// ---- POUs/Logic/Sequencing/Permissives/FB_Permissives.TcPOU
(*
PERMISSIVE - Operational Enabling Function Block
================================================
Philosophy: Allows a change in state only when all conditions are met.
Behavior:   Follows real-time conditions, no latching, can be bypassed for
            maintenance.
Logic:      Mapped bits 1 = good, 0 = bad. Unmapped bits default good (1).
            sts.bOK = TRUE when every active permissive bit is good (or
            bypassed). Non-latching: status tracks real-time inputs.
Mapping:    Call MapInput(bitIndex, value) every cycle for each active
            permissive. Unmapped bits automatically reset to good after
            FB_BitMatrix64's MAPPING_TIMEOUT cycles.

The 64-bit condition-matrix machinery is shared with FB_Interlock via
FB_BitMatrix64 — the difference between the two FBs is latching semantics,
which lives here (or in FB_Interlock) on top of the shared core.
*)
{attribute 'OPC.UA.DA' := '1'}
FUNCTION_BLOCK PUBLIC FB_Permissives
VAR_INPUT
    {attribute 'OPC.UA.DA' := '1'}
    {attribute 'OPC.UA.DA.Access' := '1'}
    cfg : ST_Permissive_Config;
END_VAR
VAR_OUTPUT
    {attribute 'OPC.UA.DA' := '1'}
    {attribute 'OPC.UA.DA.Access' := '1'}
    sts : ST_Permissive_Status;
END_VAR
VAR
    {attribute 'OPC.UA.DA' := '0'}
    _core : FB_BitMatrix64;
END_VAR

// Drive the shared bit-matrix machinery (cycle counter, cleanup, transitions).
_core.ConstrainBypass(allowedMask := cfg.nBypassable);
_core();

// Non-latching rollup: unmapped bits default good, bypassed bits forced good.
sts.nPermissives          := (_core.nLiveBits OR NOT _core.nActiveMask) OR _core.nBypassMask;
sts.nBypassMask           := _core.nBypassMask;
sts.nFirstFailureBitIndex := _core.nFirstFailureBitIndex;
sts.bOK                   := sts.nPermissives = 16#FFFFFFFFFFFFFFFF;

sts.nMissing := cfg.nRequired AND NOT _core.nActiveMask;
sts.nPermissives := sts.nPermissives AND NOT sts.nMissing;
sts.bOK := sts.bOK AND (sts.nMissing = 0);
UpdateFaceplates();

(*
Map a boolean signal to one permissive bit (0..63). TRUE = good, FALSE = bad.
Call every cycle for each active permissive condition.
*)
METHOD PUBLIC MapInput
VAR_INPUT
    bitIndex   : UDINT;
    inputValue : BOOL;
END_VAR
_core.MapInput(bitIndex := bitIndex, inputValue := inputValue);
END_METHOD

(*
Reset - Clear all bypass states. Permissives follow real-time conditions
(non-latching) so there is nothing else to clear.
*)
METHOD Reset
_core.ClearBypass();
END_METHOD

(*
Set or clear bypass for a specific permissive bit. Only bits configured
as bypassable in cfg.nBypassable can be enabled; clearing is always allowed.
*)
METHOD PUBLIC SetBypass : E_RpcMethodResponse
VAR_INPUT
    bitIndex : UDINT;
    bEnable  : BOOL;
END_VAR
SetBypass := _core.SetBypass(
    bitIndex        := bitIndex,
    bEnable         := bEnable,
    nBypassableMask := cfg.nBypassable);
END_METHOD

METHOD PRIVATE UpdateFaceplates
VAR
    i       : UDINT;
    bitMask : ULINT;
END_VAR
FOR i := 0 TO 63 DO
    bitMask := SHL(ULINT#1, i);
    sts.aFaceplates[i].name          := cfg.aNames[i];
    sts.aFaceplates[i].ok         := (sts.nPermissives AND bitMask) <> 0;
    sts.aFaceplates[i].mapped     := (_core.nActiveMask AND bitMask) <> 0;
    sts.aFaceplates[i].bypassed   := (_core.nBypassMask AND bitMask) <> 0;
    sts.aFaceplates[i].bypassable := (cfg.nBypassable  AND bitMask) <> 0;
END_FOR;
END_METHOD

END_FUNCTION_BLOCK

// ---- POUs/Utilities/FB_BitMatrix64.TcPOU
// ============================================================================
// FB_BitMatrix64 — Shared 64-bit condition-matrix core
// ============================================================================
// Internal composition helper used by FB_Permissives (non-latching) and
// FB_Interlock (latching). Encapsulates the mechanics both FBs share:
//
//   - 64 bits of "good (1) / bad (0)" live state fed by MapInput()
//   - an active-mask so unmapped bits default to good and bypass logic is
//     parameterised on the caller's cfg.nBypassable (no cfg coupling here)
//   - cycle-based cleanup that unmaps a bit if it hasn't been re-fed within
//     MAPPING_TIMEOUT scans
//   - first-failure tracking (sequence counter + first-failure bit index)
//   - "just unmapped while bad" events so the caller can latch that memory
//     if it needs to (FB_Interlock.nUnmappedBadBits)
//
// The caller composes an instance, calls the cyclic body, then computes its
// own effective mask / rollup (interlocks latch; permissives don't). See
// docs/2-Architecture.md for the split between the two surfaces.
// ============================================================================
{attribute 'OPC.UA.DA' := '0'}
FUNCTION_BLOCK FB_BitMatrix64
VAR_OUTPUT
    // Current live bits (1=good, 0=bad). Unmapped bits are held at 1.
    nLiveBits             : ULINT := 16#FFFFFFFFFFFFFFFF;
    // 1 = bit is actively mapped (refreshed within MAPPING_TIMEOUT cycles).
    nActiveMask           : ULINT := 0;
    // Dynamic bypass mask (1=bypassed). See SetBypass / ClearBypass.
    nBypassMask           : ULINT := 0;
    // Bit index (0..63) of the first bit to go bad in the current failure
    // sequence; 999 when no sequence is active.
    nFirstFailureBitIndex : UDINT := 999;
    // Bits that transitioned from active to unmapped *this cycle* while
    // their live value was bad. OR'd each cycle; caller latches if it cares.
    nJustUnmappedBad      : ULINT := 0;
END_VAR
VAR
    _previousBits     : ULINT := 16#FFFFFFFFFFFFFFFF;
    _cycleCounter     : UDINT := 0;
    _lastMappedCycle  : ARRAY[0..63] OF UDINT;
    _sequenceCounter  : UDINT := 0;
    MAPPING_TIMEOUT   : UDINT := 10;
END_VAR

_cycleCounter := _cycleCounter + 1;
IF _cycleCounter = 0 THEN _cycleCounter := 1; END_IF;

nJustUnmappedBad := 0;
_CleanupUnmapped();
_DetectTransitions();

_previousBits := nLiveBits;

// Feed one bit's live value. Call every cycle for every active condition;
// any bit not refreshed within MAPPING_TIMEOUT scans is automatically
// considered unmapped and its live bit snaps back to good.
METHOD PUBLIC MapInput
VAR_INPUT
    bitIndex   : UDINT;
    inputValue : BOOL;
END_VAR
VAR
    bitMask : ULINT;
END_VAR
IF bitIndex > 63 THEN RETURN; END_IF;

bitMask := SHL(ULINT#1, bitIndex);
nActiveMask := nActiveMask OR bitMask;
_lastMappedCycle[bitIndex] := _cycleCounter;

IF inputValue THEN
    nLiveBits := nLiveBits OR bitMask;
ELSE
    nLiveBits := nLiveBits AND NOT bitMask;
END_IF;
END_METHOD

// Enable/disable bypass for a single bit. The caller passes its own
// cfg.nBypassable so this FB stays decoupled from caller-specific cfg DUTs.
// Clearing a bypass is always permitted; enabling requires the bit to be
// marked bypassable.
METHOD PUBLIC SetBypass : E_RpcMethodResponse
VAR_INPUT
    bitIndex         : UDINT;
    bEnable          : BOOL;
    nBypassableMask  : ULINT;
END_VAR
VAR
    bitMask : ULINT;
END_VAR
IF bitIndex > 63 THEN
    SetBypass := E_RpcMethodResponse.REJECTED_INVALID_PARAMETER;
    RETURN;
END_IF;

bitMask := SHL(ULINT#1, bitIndex);

IF bEnable AND (nBypassableMask AND bitMask) = 0 THEN
    SetBypass := E_RpcMethodResponse.REJECTED_BYPASS_NOT_ALLOWED;
    RETURN;
END_IF;

IF bEnable THEN
    nBypassMask := nBypassMask OR bitMask;
ELSE
    nBypassMask := nBypassMask AND NOT bitMask;
END_IF;

SetBypass := E_RpcMethodResponse.ACCEPTED;
END_METHOD

// Clear every bypass bit at once (e.g. on a Reset()).
METHOD PUBLIC ClearBypass
nBypassMask := 0;
END_METHOD

// Drop any first-failure sequence in progress.
METHOD PUBLIC ClearFirstFailure
nFirstFailureBitIndex := 999;
_sequenceCounter      := 0;
END_METHOD

METHOD PRIVATE _CleanupUnmapped
VAR
    i       : UDINT;
    bitMask : ULINT;
END_VAR
FOR i := 0 TO 63 DO
    bitMask := SHL(ULINT#1, i);
    IF (nActiveMask AND bitMask) <> 0 THEN
        IF (_cycleCounter - _lastMappedCycle[i]) > MAPPING_TIMEOUT THEN
            // Expose bad-at-unmap as an event so latching callers (FB_Interlock)
            // can remember it. Non-latching callers simply ignore this output.
            IF (nLiveBits AND bitMask) = 0 THEN
                nJustUnmappedBad := nJustUnmappedBad OR bitMask;
            END_IF;
            nActiveMask := nActiveMask AND NOT bitMask;
            nLiveBits   := nLiveBits   OR bitMask;
        END_IF;
    END_IF;
END_FOR;
END_METHOD

METHOD PRIVATE _DetectTransitions
VAR
    i       : UDINT;
    bitMask : ULINT;
END_VAR
// New failure sequence: all-good last cycle, something bad now.
IF _previousBits = 16#FFFFFFFFFFFFFFFF AND nLiveBits <> 16#FFFFFFFFFFFFFFFF THEN
    _sequenceCounter      := 0;
    nFirstFailureBitIndex := 999;
END_IF;

FOR i := 0 TO 63 DO
    bitMask := SHL(ULINT#1, i);
    IF (nActiveMask AND bitMask) <> 0 THEN
        IF ((_previousBits AND bitMask) <> 0) AND ((nLiveBits AND bitMask) = 0) THEN
            _sequenceCounter := _sequenceCounter + 1;
            IF _sequenceCounter = 1 THEN
                nFirstFailureBitIndex := i;
            END_IF;
        END_IF;
    END_IF;
END_FOR;
END_METHOD

// Revocation is permanent; allowing the bit again requires a fresh SetBypass.
METHOD PUBLIC ConstrainBypass
VAR_INPUT allowedMask : ULINT; END_VAR
nBypassMask := nBypassMask AND allowedMask;
END_METHOD

END_FUNCTION_BLOCK

// ---- POUs/Logic/Interlocks/FB_Interlock.TcPOU
(*
INTERLOCK - Safety Protection Function Block
============================================
Philosophy: Prevents unsafe conditions from continuing. Latches bad
            conditions until a deliberate Reset() call, even if the
            real-world condition has already recovered.
Behavior:   Every mapped bit latches by design. Reset() is required to
            clear latched bits. Bypass is available per bit only if
            cfg.nBypassable marks the bit as bypassable.
Logic:      Mapped bits 1 = good, 0 = bad. Unmapped bits default good.
            A bit that was bad at the time its mapping stopped is
            remembered and keeps sts.bOK FALSE until Reset() is called.
            sts.bOK = TRUE when every active interlock bit is good.
Mapping:    Call MapInput(bitIndex, value) every cycle for each active
            interlock condition. Unmapped bits automatically reset to
            good after FB_BitMatrix64's MAPPING_TIMEOUT cycles.
Clearing:   Call Reset() after the real-world conditions have cleared.

The 64-bit condition-matrix machinery is shared with FB_Permissives via
FB_BitMatrix64; the latching + unmapped-bad memory is the interlock-only
logic that sits on top.

Contrast with FB_Permissives: permissives are non-latching operational
readiness checks; interlocks are latching safety protections.
*)
{attribute 'OPC.UA.DA' := '1'}
FUNCTION_BLOCK PUBLIC FB_Interlock
VAR_INPUT
    {attribute 'OPC.UA.DA' := '1'}
    {attribute 'OPC.UA.DA.Access' := '1'}
    cfg : ST_Interlock_Config;
END_VAR
VAR_OUTPUT
    {attribute 'OPC.UA.DA' := '1'}
    {attribute 'OPC.UA.DA.Access' := '1'}
    sts : ST_Interlock_Status;
END_VAR
VAR
    {attribute 'OPC.UA.DA' := '0'}
    _core            : FB_BitMatrix64;
    {attribute 'OPC.UA.DA' := '0'}
    _latchedBits     : ULINT := 16#FFFFFFFFFFFFFFFF;
    {attribute 'OPC.UA.DA' := '0'}
    _unmappedBadBits : ULINT := 0;
END_VAR

// Drive the shared bit-matrix machinery (cycle counter, cleanup, transitions).
_core.ConstrainBypass(allowedMask := cfg.nBypassable);
_core();

// Carry forward any "bad at unmap" memory — keeps sts.bOK FALSE until Reset().
_unmappedBadBits := _unmappedBadBits OR _core.nJustUnmappedBad OR (cfg.nRequired AND NOT _core.nActiveMask);

// Latch once a mapped bit goes bad; inactive/unmapped bits remain good.
_latchedBits := (_latchedBits AND _core.nLiveBits) OR NOT _core.nActiveMask;

// Effective: latched-or-unmapped, then forced good by any bypass bits.
sts.nInterlocks           := (_latchedBits OR NOT _core.nActiveMask) OR _core.nBypassMask;
sts.nLatched              := _latchedBits;
sts.nBypassMask           := _core.nBypassMask;
sts.nFirstFailureBitIndex := _core.nFirstFailureBitIndex;
sts.bOK                   := (sts.nInterlocks = 16#FFFFFFFFFFFFFFFF) AND (_unmappedBadBits = 0);

sts.nMissing := cfg.nRequired AND NOT _core.nActiveMask;
sts.nInterlocks := sts.nInterlocks AND NOT sts.nMissing;
sts.bOK := sts.bOK AND (sts.nMissing = 0);
UpdateFaceplates();

(*
Map a boolean input signal to a specific interlock bit (0..63).
Call every cycle for each active interlock condition.
TRUE = good / safe, FALSE = bad / unsafe.
*)
METHOD PUBLIC MapInput
VAR_INPUT
    bitIndex   : UDINT;
    inputValue : BOOL;
END_VAR
_core.MapInput(bitIndex := bitIndex, inputValue := inputValue);
END_METHOD

(*
Reset - clear latched bits by snapping them to the current live value.
Active bits that are currently good become good; active bits still bad
stay bad. Unmapped bits remain good. Also clears the unmapped-bad memory
and the first-failure sequence. Bypass states are intentionally preserved
— use SetBypass(i, FALSE) to clear them.
*)
METHOD Reset
// Snap latched bits to current live values on active bits; unmapped stay good.
_latchedBits     := (_core.nLiveBits AND _core.nActiveMask) OR NOT _core.nActiveMask;
_unmappedBadBits := 0;
_core.ClearFirstFailure();
END_METHOD

(*
Set or clear bypass for a specific interlock bit. Only bits configured as
bypassable in cfg.nBypassable can be enabled; clearing is always allowed.
WARNING: bypassing an interlock disables safety protection — use with care.
*)
METHOD PUBLIC SetBypass : E_RpcMethodResponse
VAR_INPUT
    bitIndex : UDINT;
    bEnable  : BOOL;
END_VAR
SetBypass := _core.SetBypass(
    bitIndex        := bitIndex,
    bEnable         := bEnable,
    nBypassableMask := cfg.nBypassable);
END_METHOD

METHOD PRIVATE UpdateFaceplates
VAR
    i       : UDINT;
    bitMask : ULINT;
END_VAR
FOR i := 0 TO 63 DO
    bitMask := SHL(ULINT#1, i);
    sts.aFaceplates[i].name          := cfg.aNames[i];
    sts.aFaceplates[i].ok         := (sts.nInterlocks AND bitMask) <> 0;
    sts.aFaceplates[i].live       := (_core.nLiveBits  AND bitMask) <> 0;
    sts.aFaceplates[i].latched    := ((_core.nActiveMask AND bitMask) <> 0) AND ((_latchedBits AND bitMask) = 0);
    sts.aFaceplates[i].mapped     := (_core.nActiveMask AND bitMask) <> 0;
    sts.aFaceplates[i].bypassed   := (_core.nBypassMask AND bitMask) <> 0;
    sts.aFaceplates[i].bypassable := (cfg.nBypassable   AND bitMask) <> 0;
END_FOR;
END_METHOD

END_FUNCTION_BLOCK

// ---- POUs/Logic/Sequencing/StateMachine/FB_StateMachine.TcPOU
FUNCTION_BLOCK FB_StateMachine EXTENDS FB_DeviceBase
VAR_INPUT
    cfgAutoRun : BOOL;
    inpShutdownConfirmed : BOOL; // Application confirmation required to reset a failed Abort.
    cfgHome : ST_Permissive_Config;
    cfgStart : ST_Permissive_Config;
    cfgProceed : ST_Permissive_Config;
    cfgAuto : ST_Permissive_Config;
    cfgRunning : ST_Interlock_Config;
    inpSubmoduleFaulted : BOOL;
END_VAR

VAR_OUTPUT
    Status : ST_SM_Status;
END_VAR

VAR CONSTANT
    HOMING_MIN   : DINT := 1000; HOMING_MAX   : DINT := 1999;
    RUNNING_MIN  : DINT := 3000; RUNNING_MAX  : DINT := 3999;
    STOPPING_MIN : DINT := 2000; STOPPING_MAX : DINT := 2999;
    ABORTING_MIN : DINT := 5000; ABORTING_MAX : DINT := 5999;
    PAUSING_MIN  : DINT := 4000; PAUSING_MAX  : DINT := 4999;
    PROCEEDING_MIN : DINT := 6000; PROCEEDING_MAX : DINT := 6999;
END_VAR

VAR
    // Internal command request flags (set by methods, consumed by body)
    _abortRequested : BOOL;
    _completeStateRequested : BOOL;
    _homeRequested : BOOL;
    _pauseRequested : BOOL;
    _proceedRequested : BOOL;
    _startRequested : BOOL;
    _stopRequested : BOOL;
    _retryActive : BOOL;
    RetryComplete : BOOL;

    // OEE condition latches. Updated by ReportBlocked / ReportStarved, consumed
    // and cleared by the body each cycle. Kept internal so the FB contract
    // never mutates external inputs.
    _blockedCode : DINT;
    _starvedCode : DINT;

    // Timer
    StepTimer : TON;

    // Edge detection
    R_TRIG_1 : R_TRIG;

    // Internal state tracking
    _previousState : E_SM_State;
    PreviousStep : DINT;
    TimerReset : BOOL;
    LsOdd : DINT;
    _returnState : E_SM_State;
    ReturnNextStep : DINT;

    // Permission handlers
    permAuto : FB_Permissives;
    permHome : FB_Permissives;
    permProceed : FB_Permissives;
    permStart : FB_Permissives;

    // Running interlock (latching - auto-aborts from any active state)
    intlkRunning : FB_Interlock;

    // Step ownership (internal)
    _nextStep : DINT;
    _coverageStep : DINT := -1;
    _activeStepCalls : UINT;
    _stepFailurePending : BOOL;
    _stepRecoveryPending : BOOL;
END_VAR

_ProcessOperatorCommands();

//-----------------------------------------------------------------------------
// Main Implementation
//-----------------------------------------------------------------------------
//-------------------------------------------------------------------------
// Process permissions for different states
//-------------------------------------------------------------------------
permHome(cfg := cfgHome);
permStart(cfg := cfgStart);
permProceed(cfg := cfgProceed);
permAuto(cfg := cfgAuto);

intlkRunning(cfg := cfgRunning);
    IF inpSubmoduleFaulted THEN
        _Raise(
            code   := E_SM_Fault.SubmoduleFaulted,
            source := 'SUBMODULE',
            reason := 'Submodule reported fault via inpSubmoduleFaulted'
        );
    END_IF;
IF inpSubmoduleFaulted AND Status.State <> E_SM_State.STOPPED AND Status.State <> E_SM_State.ABORTING THEN _abortRequested := TRUE; END_IF;


    // Auto-abort if any running interlock trips (e-stop, safety gate, etc.)
    IF NOT intlkRunning.sts.bOK AND
       NOT (Status.State = E_SM_State.STOPPED OR Status.State = E_SM_State.ABORTING) THEN
        _abortRequested := TRUE;
        _Raise(
            code   := E_SM_Fault.RunningInterlockTripped,
            source := 'INTLK_RUNNING',
            reason := 'Running interlock tripped, auto-aborting'
        );
    END_IF;

    // Observe the completed application scan before consuming another transition.
    IF _coverageStep = Status.Step.Current AND Status.ActiveState AND
       Status.Step.Current MOD 2 = 0 AND NOT _stepFailurePending AND
       (NOT IsFaulted() OR Status.State = E_SM_State.STOPPING OR Status.State = E_SM_State.ABORTING) THEN
        IF _activeStepCalls = 0 THEN
            _RaiseStepFault(stepNum := Status.Step.Current, stepName := Status.Step.Name,
                code := E_SM_Fault.MissingStepImplementation, reason := 'Active FB_Step was not called in the application scan');
        ELSIF _activeStepCalls > 1 THEN
            _RaiseStepFault(stepNum := Status.Step.Current, stepName := Status.Step.Name,
                code := E_SM_Fault.DuplicateStepImplementation, reason := 'Active step was executed more than once in the application scan');
        END_IF;
    END_IF;
    _activeStepCalls := 0;

    _previousState := Status.State;
    // Sequence completion is a zero next-step requested from a valid active step.
    _completeStateRequested := _IsStepInStateRange(state := Status.State, nStep := Status.Step.Current) AND _nextStep = 0;
    Status.AutoCycleRequest := cfgAutoRun AND Status.State = E_SM_State.READY AND Status.LastState = E_SM_State.RUNNING AND NOT permStart.sts.bOK;

    // One transition per scan. Abort > Stop > fault recovery > normal transition.
    IF _stepFailurePending AND Status.State = E_SM_State.ABORTING THEN
        Status.State := E_SM_State.STOPPED;
        Status.ShutdownFailed := TRUE;
        _Raise(code := E_SM_Fault.ShutdownFailed, source := 'ABORT', reason := 'Abort sequence failed; physical shutdown confirmation required');
    ELSIF _abortRequested OR (_stepFailurePending AND Status.State = E_SM_State.STOPPING) THEN
        IF Status.State <> E_SM_State.STOPPED AND Status.State <> E_SM_State.ABORTING THEN
            Status.State := E_SM_State.ABORTING;
        END_IF;
    ELSIF _stopRequested THEN
        IF Status.State = E_SM_State.READY THEN
            Status.State := E_SM_State.STOPPED;
        ELSIF Status.State <> E_SM_State.STOPPED AND Status.State <> E_SM_State.ABORTING THEN
            Status.State := E_SM_State.STOPPING;
        END_IF;
    ELSE
        CASE Status.State OF
            E_SM_State.STOPPED:
                IF _homeRequested AND NOT IsFaulted() AND permHome.sts.bOK AND permAuto.sts.bOK AND intlkRunning.sts.bOK THEN
                    Status.State := E_SM_State.HOMING;
                END_IF;
            E_SM_State.READY:
                IF (_startRequested OR (cfgAutoRun AND Status.LastState = E_SM_State.RUNNING)) AND NOT IsFaulted() AND permStart.sts.bOK AND permAuto.sts.bOK AND intlkRunning.sts.bOK THEN
                    Status.State := E_SM_State.RUNNING;
                END_IF;
            E_SM_State.HOMING, E_SM_State.RUNNING:
                IF NOT IsFaulted() THEN
                    IF _pauseRequested AND Status.State = E_SM_State.RUNNING THEN
                        _returnState := Status.State;
                        ReturnNextStep := Status.Step.Current;
                        Status.State := E_SM_State.PAUSING;
                    ELSIF _completeStateRequested THEN
                        Status.State := E_SM_State.READY;
                    END_IF;
                END_IF;
            E_SM_State.PAUSING:
                IF _completeStateRequested AND NOT IsFaulted() THEN Status.State := E_SM_State.PAUSED; END_IF;
            E_SM_State.PAUSED:
                IF _proceedRequested AND NOT IsFaulted() AND permProceed.sts.bOK AND permAuto.sts.bOK AND intlkRunning.sts.bOK THEN
                    Status.State := E_SM_State.PROCEEDING;
                END_IF;
            E_SM_State.PROCEEDING:
                IF _completeStateRequested AND NOT IsFaulted() THEN Status.State := _returnState; END_IF;
            E_SM_State.STOPPING, E_SM_State.ABORTING:
                IF _completeStateRequested THEN Status.State := E_SM_State.STOPPED; END_IF;
        END_CASE;
    END_IF;
    IF Status.State <> _previousState THEN
        _stepFailurePending := FALSE;
        _stepRecoveryPending := FALSE;
        _ClearStepPermissives();
        Status.Step.Name := '';
        IF _previousState = E_SM_State.PROCEEDING AND Status.State = _returnState THEN
            _nextStep := ReturnNextStep;
        ELSE
            _nextStep := _GetFirstStepForState(state := Status.State);
        END_IF;
    END_IF;

    //-------------------------------------------------------------------------
    // Track state changes
    //-------------------------------------------------------------------------
    IF Status.State <> _previousState THEN
        Status.LastState := _previousState;
    END_IF;

    //-------------------------------------------------------------------------
    // Derived status flags
    //-------------------------------------------------------------------------
    Status.WaitingState := (Status.State = E_SM_State.STOPPED) OR (Status.State = E_SM_State.READY) OR
                           (Status.State = E_SM_State.PAUSED);
    Status.ActiveState  := (Status.State = E_SM_State.HOMING) OR (Status.State = E_SM_State.RUNNING) OR
                           (Status.State = E_SM_State.STOPPING) OR (Status.State = E_SM_State.PAUSING) OR
                           (Status.State = E_SM_State.PROCEEDING) OR (Status.State = E_SM_State.ABORTING);

    //-------------------------------------------------------------------------
    // Step and timer management
    //-------------------------------------------------------------------------

    // Reset timer and clear step name when transitioning to step 0
    R_TRIG_1(CLK := Status.Step.Current = 0);
    IF R_TRIG_1.Q THEN
        Status.Step.Name := '';
        _ClearStepPermissives();
        TimerReset := TRUE;
        StepTimer(IN := FALSE, PT := T#99H);
        Status.Step.TimerSeconds := 0.0;
    END_IF;

    // Auto-initialize first step when entering an active state
    IF Status.Step.Current = 0 AND Status.ActiveState THEN
        _nextStep := _GetFirstStepForState(state := Status.State);
    END_IF;

    // Detect step change and update
    IF Status.Step.Current <> _nextStep THEN
        PreviousStep := Status.Step.Current;
        Status.Step.Current := _nextStep;
        TimerReset := TRUE;
        StepTimer(IN := FALSE, PT := T#99H);
        Status.Step.TimerSeconds := 0.0;
    END_IF;

    Status.Step.Next := _nextStep;

    // Step timer logic
    IF NOT (Status.State = E_SM_State.PAUSED) OR ((Status.State = E_SM_State.PAUSED) AND _completeStateRequested) THEN
        IF TimerReset THEN
            StepTimer(IN := FALSE, PT := T#99H);
            Status.Step.TimerSeconds := 0.0;
            TimerReset := FALSE;
        ELSE
            StepTimer(IN := TRUE, PT := T#99H);
            Status.Step.TimerSeconds := UDINT_TO_REAL(TIME_TO_UDINT(StepTimer.ET)) / 1000.0;
        END_IF;
    ELSE
        StepTimer(IN := FALSE, PT := T#99H);
    END_IF;

    //-------------------------------------------------------------------------
    // Fault detection â€” surface through the shared fault handler so the
    // ring-buffer/history in ST_DeviceHeader_Sts stays populated.
    //
    // Ordering discipline:
    //   1. Submodule faults raise immediately with a specific code + source.
    //   2. OddStepReached is the "nothing more specific said anything" default
    //      for landing on an odd step. We only auto-raise it when no fault is
    //      currently active, so a more specific raise (StepTimeout raised by
    //      FB_Step, StepUserFault raised by step.RaiseFault, etc.) wins.
    //-------------------------------------------------------------------------
    LsOdd := Status.Step.Current MOD 2;
    Status.AtRecoveryStep := LsOdd <> 0;
    Status.SubmoduleFaulted := inpSubmoduleFaulted;



    IF Status.AtRecoveryStep AND GetFaultCode() = 0 THEN
        _RaiseStepFault(
            stepNum  := Status.Step.Current,
            stepName := Status.Step.Name,
            code     := E_SM_Fault.OddStepReached,
            reason   := ''
        );
    END_IF;

    //-------------------------------------------------------------------------
    // Retry logic
    //-------------------------------------------------------------------------
    IF RetryComplete THEN
        _retryActive := FALSE;
        RetryComplete := FALSE;
    END_IF;

    IF _retryActive THEN
        RetryComplete := TRUE;
    END_IF;

    IF _retryActive AND Status.AtRecoveryStep AND NOT _abortRequested AND NOT _stopRequested THEN
        // Roll back to previous (even, non-faulted) step to re-enter it
        IF NOT inpSubmoduleFaulted AND intlkRunning.sts.bOK THEN
            _ClearFault();
            _stepFailurePending := FALSE;
            _stepRecoveryPending := FALSE;
            _nextStep := Status.Step.Current - 1;
        END_IF;
    END_IF;

    //-------------------------------------------------------------------------
    // OEE condition codes (Blocked / Starved) â€” consume the internal latches.
    // The latches are fed externally via ReportBlocked() / ReportStarved().
    //-------------------------------------------------------------------------
    IF _blockedCode = 0 THEN
        Status.BlockedCondition := 0;
    END_IF;

    IF _blockedCode <> 0 AND
       (Status.State = E_SM_State.RUNNING OR Status.State = E_SM_State.STOPPING OR
        Status.State = E_SM_State.READY) THEN
        Status.BlockedCondition := _blockedCode;
        _blockedCode := 0;
    END_IF;

    IF _starvedCode = 0 THEN
        Status.StarvedCondition := 0;
    END_IF;

    IF _starvedCode <> 0 AND
       (Status.State = E_SM_State.RUNNING OR Status.State = E_SM_State.STOPPING OR
        Status.State = E_SM_State.READY) THEN
        Status.StarvedCondition := _starvedCode;
        _starvedCode := 0;
    END_IF;

    //-------------------------------------------------------------------------
    // Common device header (stateString, ready/Busy/Faulted/SourceLocked,
    // fault codes + strings, timestamps). Published via Status.header.
    //-------------------------------------------------------------------------
    Status.Faulted := IsFaulted();
    Status.ReadyToHome := Status.State = E_SM_State.STOPPED AND NOT IsFaulted() AND permHome.sts.bOK AND permAuto.sts.bOK AND intlkRunning.sts.bOK;
    Status.ReadyToStart := Status.State = E_SM_State.READY AND NOT IsFaulted() AND permStart.sts.bOK AND permAuto.sts.bOK AND intlkRunning.sts.bOK;
    Status.ReadyToProceed := Status.State = E_SM_State.PAUSED AND NOT IsFaulted() AND permProceed.sts.bOK AND permAuto.sts.bOK AND intlkRunning.sts.bOK;
    _coverageStep := Status.Step.Current;
    _ClearCommandFlags();
    _UpdateHeader(
        header      := Status.header,
        stateString := _StateToString(state := Status.State),
        busy     := Status.ActiveState
    );

METHOD PRIVATE _ClearStepPermissives
VAR
    i : UDINT;
END_VAR
Status.Step.PermCfg.nRequired := 0;
Status.Step.PermCfg.nBypassable := 0;
Status.Step.PermStatus.bOK := FALSE;
Status.Step.PermStatus.nPermissives := 0;
Status.Step.PermStatus.nBypassMask := 0;
Status.Step.PermStatus.nFirstFailureBitIndex := 999;

FOR i := 0 TO 63 DO
    Status.Step.PermCfg.aNames[i]                       := '';
    Status.Step.PermStatus.aFaceplates[i].name          := '';
    Status.Step.PermStatus.aFaceplates[i].ok         := FALSE;
    Status.Step.PermStatus.aFaceplates[i].mapped     := FALSE;
    Status.Step.PermStatus.aFaceplates[i].bypassed   := FALSE;
    Status.Step.PermStatus.aFaceplates[i].bypassable := FALSE;
END_FOR;
END_METHOD

METHOD PRIVATE _GetFirstStepForState : DINT
VAR_INPUT
        state : E_SM_State;
END_VAR
CASE state OF
        E_SM_State.HOMING:     _GetFirstStepForState := HOMING_MIN;
        E_SM_State.RUNNING:    _GetFirstStepForState := RUNNING_MIN;
        E_SM_State.STOPPING:   _GetFirstStepForState := STOPPING_MIN;
        E_SM_State.ABORTING:   _GetFirstStepForState := ABORTING_MIN;
        E_SM_State.PAUSING:    _GetFirstStepForState := PAUSING_MIN;
        E_SM_State.PROCEEDING: _GetFirstStepForState := PROCEEDING_MIN;
ELSE
        _GetFirstStepForState := 0;
END_CASE;
END_METHOD

METHOD PRIVATE _GetLastStepForState : DINT
VAR_INPUT
        state : E_SM_State;
END_VAR
CASE state OF
        E_SM_State.HOMING:     _GetLastStepForState := HOMING_MAX;
        E_SM_State.RUNNING:    _GetLastStepForState := RUNNING_MAX;
        E_SM_State.STOPPING:   _GetLastStepForState := STOPPING_MAX;
        E_SM_State.ABORTING:   _GetLastStepForState := ABORTING_MAX;
        E_SM_State.PAUSING:    _GetLastStepForState := PAUSING_MAX;
        E_SM_State.PROCEEDING: _GetLastStepForState := PROCEEDING_MAX;
ELSE
        _GetLastStepForState := 0;
END_CASE;
END_METHOD

METHOD PRIVATE _IsStepInStateRange : BOOL
VAR_INPUT
        state : E_SM_State;
        nStep : DINT;
END_VAR
_IsStepInStateRange := (_GetFirstStepForState(state := state) > 0) AND (nStep >= _GetFirstStepForState(state := state)) AND
                                             (nStep <= _GetLastStepForState(state := state));
END_METHOD

METHOD PRIVATE _StateToString : STRING(31)
VAR_INPUT
    state : E_SM_State;
END_VAR
CASE state OF
    E_SM_State.STOPPED:    _StateToString := 'STOPPED';
    E_SM_State.READY:      _StateToString := 'READY';
    E_SM_State.PAUSED:     _StateToString := 'PAUSED';
    E_SM_State.HOMING:     _StateToString := 'HOMING';
    E_SM_State.RUNNING:    _StateToString := 'RUNNING';
    E_SM_State.STOPPING:   _StateToString := 'STOPPING';
    E_SM_State.ABORTING:   _StateToString := 'ABORTING';
    E_SM_State.PAUSING:    _StateToString := 'PAUSING';
    E_SM_State.PROCEEDING: _StateToString := 'PROCEEDING';
ELSE
    _StateToString := 'UNKNOWN';
END_CASE;
END_METHOD

// Reset every pending command-request flag. Each public command method
// calls this first, then re-sets the single flag it actually requests, so
// the body only ever sees one active request at a time.
METHOD PRIVATE _ClearCommandFlags
_abortRequested         := FALSE;
_completeStateRequested := FALSE;
_homeRequested          := FALSE;
_pauseRequested         := FALSE;
_proceedRequested       := FALSE;
_startRequested         := FALSE;
_stopRequested          := FALSE;
END_METHOD

METHOD PROTECTED ResolveFaultString : STRING(79)
VAR_INPUT
    code : DINT;
END_VAR
CASE code OF
    E_SM_Fault.InvalidStepConfiguration: ResolveFaultString := 'Invalid Step Configuration';
    E_SM_Fault.MissingStepImplementation: ResolveFaultString := 'Missing Step Implementation';
    E_SM_Fault.DuplicateStepImplementation: ResolveFaultString := 'Duplicate Step Implementation';
    E_SM_Fault.ShutdownFailed: ResolveFaultString := 'Shutdown Failed';
    E_SM_Fault.None:                    ResolveFaultString := 'No Fault';
    E_SM_Fault.StepTimeout:             ResolveFaultString := 'Step Timeout';
    E_SM_Fault.OddStepReached:          ResolveFaultString := 'Step Faulted';
    E_SM_Fault.StepUserFault:           ResolveFaultString := 'Step User Fault';
    E_SM_Fault.RunningInterlockTripped: ResolveFaultString := 'Running Interlock Tripped';
    E_SM_Fault.SubmoduleFaulted:        ResolveFaultString := 'Submodule Faulted';
ELSE
    ResolveFaultString := 'Unknown Fault';
END_CASE;
END_METHOD

// Safety command â€” always accepted (bypasses source lock and fault check).
// Rejected only when the machine is already terminally stopped or already
// running the Abort sequence.
METHOD Abort : E_RpcMethodResponse
VAR_INPUT
    eRequester : E_Requester := E_Requester.PROG;
END_VAR
// Reject invalid identity before any command-specific mutation.
Abort := F_ValidateRequester(eRequester := eRequester, bSourceLocked := FALSE, bFaulted := FALSE);
IF Abort <> E_RpcMethodResponse.ACCEPTED THEN RETURN; END_IF;
IF (Status.State = E_SM_State.STOPPED AND NOT _homeRequested) OR Status.State = E_SM_State.ABORTING THEN
    Abort := E_RpcMethodResponse.REJECTED_WRONG_STATE;
    RETURN;
END_IF;

_operatorMailbox.CancelNormal();
_ClearCommandFlags();
_abortRequested := TRUE;
_retryActive := FALSE;
_AcceptCommand(eRequester := eRequester);
Abort := E_RpcMethodResponse.ACCEPTED;
END_METHOD

METHOD Home : E_RpcMethodResponse
VAR_INPUT
    eRequester : E_Requester := E_Requester.PROG;
END_VAR
// Reject invalid identity before any command-specific mutation.
Home := F_ValidateRequester(eRequester := eRequester, bSourceLocked := FALSE, bFaulted := FALSE);
IF Home <> E_RpcMethodResponse.ACCEPTED THEN RETURN; END_IF;
IF _abortRequested OR _stopRequested OR _homeRequested OR _startRequested OR _pauseRequested OR _proceedRequested THEN
    Home := E_RpcMethodResponse.REJECTED_WRONG_STATE;
    RETURN;
END_IF;
Home := F_ValidateRequester(eRequester, bSourceLockedToProg, IsFaulted());
IF Home <> E_RpcMethodResponse.ACCEPTED THEN RETURN; END_IF;

IF NOT (Status.State = E_SM_State.STOPPED) THEN
    Home := E_RpcMethodResponse.REJECTED_WRONG_STATE;
    RETURN;
END_IF;

IF NOT permHome.sts.bOK THEN
    Home := E_RpcMethodResponse.REJECTED_PERMISSIVE_NOT_MET;
    RETURN;
END_IF;

IF NOT permAuto.sts.bOK THEN
    Home := E_RpcMethodResponse.REJECTED_PERMISSIVE_NOT_MET;
    RETURN;
END_IF;

_ClearCommandFlags();
_homeRequested := TRUE;
_AcceptCommand(eRequester := eRequester);
Home := E_RpcMethodResponse.ACCEPTED;
END_METHOD

METHOD Pause : E_RpcMethodResponse
VAR_INPUT
    eRequester : E_Requester := E_Requester.PROG;
END_VAR
// Reject invalid identity before any command-specific mutation.
Pause := F_ValidateRequester(eRequester := eRequester, bSourceLocked := FALSE, bFaulted := FALSE);
IF Pause <> E_RpcMethodResponse.ACCEPTED THEN RETURN; END_IF;
IF _abortRequested OR _stopRequested OR _homeRequested OR _startRequested OR _pauseRequested OR _proceedRequested THEN
    Pause := E_RpcMethodResponse.REJECTED_WRONG_STATE;
    RETURN;
END_IF;
Pause := F_ValidateRequester(eRequester, bSourceLockedToProg, IsFaulted());
IF Pause <> E_RpcMethodResponse.ACCEPTED THEN RETURN; END_IF;

IF NOT (Status.State = E_SM_State.RUNNING) THEN
    Pause := E_RpcMethodResponse.REJECTED_WRONG_STATE;
    RETURN;
END_IF;

_ClearCommandFlags();
_pauseRequested := TRUE;
_AcceptCommand(eRequester := eRequester);
Pause := E_RpcMethodResponse.ACCEPTED;
END_METHOD

METHOD Proceed : E_RpcMethodResponse
VAR_INPUT
    eRequester : E_Requester := E_Requester.PROG;
END_VAR
// Reject invalid identity before any command-specific mutation.
Proceed := F_ValidateRequester(eRequester := eRequester, bSourceLocked := FALSE, bFaulted := FALSE);
IF Proceed <> E_RpcMethodResponse.ACCEPTED THEN RETURN; END_IF;
IF _abortRequested OR _stopRequested OR _homeRequested OR _startRequested OR _pauseRequested OR _proceedRequested THEN
    Proceed := E_RpcMethodResponse.REJECTED_WRONG_STATE;
    RETURN;
END_IF;
Proceed := F_ValidateRequester(eRequester, bSourceLockedToProg, IsFaulted());
IF Proceed <> E_RpcMethodResponse.ACCEPTED THEN RETURN; END_IF;

IF NOT (Status.State = E_SM_State.PAUSED) THEN
    Proceed := E_RpcMethodResponse.REJECTED_WRONG_STATE;
    RETURN;
END_IF;

IF NOT permProceed.sts.bOK THEN
    Proceed := E_RpcMethodResponse.REJECTED_PERMISSIVE_NOT_MET;
    RETURN;
END_IF;

IF NOT permAuto.sts.bOK THEN
    Proceed := E_RpcMethodResponse.REJECTED_PERMISSIVE_NOT_MET;
    RETURN;
END_IF;

_ClearCommandFlags();
_proceedRequested := TRUE;
_AcceptCommand(eRequester := eRequester);
Proceed := E_RpcMethodResponse.ACCEPTED;
END_METHOD

METHOD Retry : E_RpcMethodResponse
VAR_INPUT
    eRequester : E_Requester := E_Requester.PROG;
END_VAR
// Reject invalid identity before any command-specific mutation.
Retry := F_ValidateRequester(eRequester := eRequester, bSourceLocked := FALSE, bFaulted := FALSE);
IF Retry <> E_RpcMethodResponse.ACCEPTED THEN RETURN; END_IF;
// Recovery bypasses the fault gate, but never source arbitration or active interlocks.
Retry := F_ValidateRequester(eRequester, bSourceLockedToProg, FALSE);
IF Retry <> E_RpcMethodResponse.ACCEPTED THEN RETURN; END_IF;
IF _abortRequested OR _stopRequested OR NOT Status.AtRecoveryStep OR
   NOT (_stepRecoveryPending OR GetFaultCode() = E_SM_Fault.OddStepReached OR GetFaultCode() = E_SM_Fault.StepTimeout OR GetFaultCode() = E_SM_Fault.StepUserFault) THEN
    Retry := E_RpcMethodResponse.REJECTED_WRONG_STATE;
    RETURN;
END_IF;
IF inpSubmoduleFaulted OR NOT intlkRunning.sts.bOK THEN
    Retry := E_RpcMethodResponse.REJECTED_INTERLOCKED;
    RETURN;
END_IF;
_retryActive := TRUE;
_AcceptCommand(eRequester := eRequester);
Retry := E_RpcMethodResponse.ACCEPTED;
END_METHOD

METHOD Start : E_RpcMethodResponse
VAR_INPUT
    eRequester : E_Requester := E_Requester.PROG;
END_VAR
// Reject invalid identity before any command-specific mutation.
Start := F_ValidateRequester(eRequester := eRequester, bSourceLocked := FALSE, bFaulted := FALSE);
IF Start <> E_RpcMethodResponse.ACCEPTED THEN RETURN; END_IF;
IF _abortRequested OR _stopRequested OR _homeRequested OR _startRequested OR _pauseRequested OR _proceedRequested THEN
    Start := E_RpcMethodResponse.REJECTED_WRONG_STATE;
    RETURN;
END_IF;
Start := F_ValidateRequester(eRequester, bSourceLockedToProg, IsFaulted());
IF Start <> E_RpcMethodResponse.ACCEPTED THEN RETURN; END_IF;

IF NOT (Status.State = E_SM_State.READY) THEN
    Start := E_RpcMethodResponse.REJECTED_WRONG_STATE;
    RETURN;
END_IF;

IF NOT permStart.sts.bOK THEN
    Start := E_RpcMethodResponse.REJECTED_PERMISSIVE_NOT_MET;
    RETURN;
END_IF;

IF NOT permAuto.sts.bOK THEN
    Start := E_RpcMethodResponse.REJECTED_PERMISSIVE_NOT_MET;
    RETURN;
END_IF;

_ClearCommandFlags();
_startRequested := TRUE;
_AcceptCommand(eRequester := eRequester);
Start := E_RpcMethodResponse.ACCEPTED;
END_METHOD

// Safety-adjacent command â€” skip source check and fault check. Rejected only
// when the machine is already terminally stopped or already stopping.
METHOD Stop : E_RpcMethodResponse
VAR_INPUT
    eRequester : E_Requester := E_Requester.PROG;
END_VAR
// Reject invalid identity before any command-specific mutation.
Stop := F_ValidateRequester(eRequester := eRequester, bSourceLocked := FALSE, bFaulted := FALSE);
IF Stop <> E_RpcMethodResponse.ACCEPTED THEN RETURN; END_IF;
IF _abortRequested OR Status.State = E_SM_State.ABORTING OR (Status.State = E_SM_State.STOPPED AND NOT _homeRequested) OR Status.State = E_SM_State.STOPPING THEN
    Stop := E_RpcMethodResponse.REJECTED_WRONG_STATE;
    RETURN;
END_IF;

_operatorMailbox.CancelNormal();
_ClearCommandFlags();
_stopRequested := TRUE;
_retryActive := FALSE;
_AcceptCommand(eRequester := eRequester);
Stop := E_RpcMethodResponse.ACCEPTED;
END_METHOD

// External hook for OEE condition reporting. Pass a non-zero reason code while
// the machine is blocked (e.g. downstream buffer full); pass 0 to clear. The
// body publishes the active code on Status.BlockedCondition in active states.
METHOD PUBLIC ReportBlocked
VAR_INPUT
    code : DINT;
END_VAR
_blockedCode := code;
END_METHOD

// External hook for OEE condition reporting. Pass a non-zero reason code while
// the machine is starved (e.g. upstream feeder empty); pass 0 to clear.
METHOD PUBLIC ReportStarved
VAR_INPUT
    code : DINT;
END_VAR
_starvedCode := code;
END_METHOD

// Map a running interlock bit. Call every cycle. bGood=TRUE means the condition is safe.
// If bGood goes FALSE from any non-stopped state the machine auto-aborts.
METHOD MapRunningIntlk
VAR_INPUT
    bitIndex : UDINT;
    bGood    : BOOL;
END_VAR
intlkRunning.MapInput(bitIndex := bitIndex, inputValue := bGood);
END_METHOD

// Clear latched running interlock bits after the real-world condition has recovered.
// The machine will still be in STOPPED/ABORTING â€” issue Home/Start separately.
METHOD ResetRunningIntlk
intlkRunning.Reset();
END_METHOD

// INTERNAL: used by FB_Step to advance the sequence. Not part of the user API.
METHOD INTERNAL SetNextStep
VAR_INPUT
    nStep : DINT;
END_VAR
IF NOT CanExecuteStep(nStep := Status.Step.Current) THEN RETURN; END_IF;
IF nStep <> 0 AND (NOT _IsStepInStateRange(state := Status.State, nStep := nStep) OR nStep MOD 2 <> 0 OR nStep = Status.Step.Current) THEN
    _RaiseStepFault(stepNum := Status.Step.Current, stepName := Status.Step.Name,
        code := E_SM_Fault.InvalidStepConfiguration, reason := 'Destination must be zero or a different even step in the same state');
    RETURN;
END_IF;
_nextStep := nStep;
END_METHOD

// INTERNAL: used by FB_Step to publish its name to StepInfo. Not part of the user API.
METHOD INTERNAL SetStepName
VAR_INPUT
    sName : STRING(40);
END_VAR
Status.Step.Name := sName;
END_METHOD

// INTERNAL: used by FB_Step to publish the active step permissive data for HMI / OPC.
METHOD INTERNAL SetStepPermissives
VAR_INPUT
        cfg : ST_Permissive_Config;
        sts : ST_Permissive_Status;
END_VAR
Status.Step.PermCfg := cfg;
Status.Step.PermStatus := sts;
END_METHOD

// INTERNAL: unified step-fault entry point used by FB_Step (timeout, user
// RaiseFault) and by the SM body (OddStepReached auto-raise). Builds a
// default reason when the caller leaves it empty so the ring never stores
// blank context, then raises through the inherited fault book-keeping.
//
// Records the failure and selects recovery or shutdown escalation.
METHOD INTERNAL _RaiseStepFault
VAR_INPUT
    stepNum  : DINT;
    stepName : STRING(40);
    code     : DINT;
    reason   : STRING(79);
END_VAR
VAR
    effectiveCode : DINT;
    srcStr    : STRING(31);
    reasonStr : STRING(79);
END_VAR
effectiveCode := code;
IF effectiveCode <= 0 THEN effectiveCode := E_SM_Fault.StepUserFault; END_IF;
srcStr := CONCAT(STR1 := 'STEP_', STR2 := DINT_TO_STRING(stepNum));

IF reason <> '' THEN
    reasonStr := reason;
ELSE
    // Default: "Step 3004 [Advance cylinder]: Step Faulted"
    reasonStr := CONCAT(STR1 := 'Step ', STR2 := DINT_TO_STRING(stepNum));
    IF stepName <> '' THEN
        reasonStr := CONCAT(STR1 := reasonStr, STR2 := ' [');
        reasonStr := CONCAT(STR1 := reasonStr, STR2 := stepName);
        reasonStr := CONCAT(STR1 := reasonStr, STR2 := ']');
    END_IF;
    reasonStr := CONCAT(STR1 := reasonStr, STR2 := ': ');
    reasonStr := CONCAT(STR1 := reasonStr, STR2 := THIS^.ResolveFaultString(code := effectiveCode));
END_IF;

_Raise(
    code   := effectiveCode,
    source := srcStr,
    reason := reasonStr
);
Status.FailedStep := stepNum;
_stepFailurePending := TRUE;
_stepRecoveryPending := Status.State <> E_SM_State.STOPPING AND Status.State <> E_SM_State.ABORTING;
IF Status.State = E_SM_State.ABORTING THEN Status.ShutdownFailed := TRUE; END_IF;
IF _stepRecoveryPending THEN
    _nextStep := stepNum;
    IF stepNum MOD 2 = 0 THEN _nextStep := stepNum + 1; END_IF;
END_IF;
END_METHOD

METHOD PUBLIC Reset : E_RpcMethodResponse
VAR_INPUT
    eRequester : E_Requester := E_Requester.PROG;
END_VAR
// Validate identity before changing any sequence recovery state. Reset bypasses source locks.
Reset := F_ValidateRequester(eRequester := eRequester, bSourceLocked := FALSE, bFaulted := FALSE);
IF Reset <> E_RpcMethodResponse.ACCEPTED THEN RETURN; END_IF;
// Reset is recovery, not a motion-stop command. Abort/Stop first.
IF Status.State <> E_SM_State.STOPPED THEN
    Reset := E_RpcMethodResponse.REJECTED_WRONG_STATE;
    RETURN;
END_IF;
IF inpSubmoduleFaulted OR NOT intlkRunning.sts.bOK THEN
    Reset := E_RpcMethodResponse.REJECTED_INTERLOCKED;
    RETURN;
END_IF;
IF Status.ShutdownFailed AND NOT inpShutdownConfirmed THEN
    Reset := E_RpcMethodResponse.REJECTED_INTERLOCKED;
    RETURN;
END_IF;
_operatorMailbox.CancelNormal();
_stepFailurePending := FALSE;
_stepRecoveryPending := FALSE;
Status.ShutdownFailed := FALSE;
Status.FailedStep := 0;
_coverageStep := -1;
_activeStepCalls := 0;
_ClearCommandFlags();
_retryActive := FALSE;
RetryComplete := FALSE;
_nextStep := 0;
Status.Step.Current := 0;
Status.AtRecoveryStep := FALSE;
Status.Faulted := FALSE;
Reset := SUPER^.Reset(eRequester := eRequester);
END_METHOD

{attribute 'TcRpcEnable' := '1'}
METHOD PUBLIC OperatorAbort : E_RpcMethodResponse

VAR_INPUT requestId : ULINT; END_VAR
OperatorAbort := _operatorMailbox.Submit(requestId := requestId, command := E_OperatorCommand.Abort, value := 0.0);
END_METHOD

{attribute 'TcRpcEnable' := '1'}
METHOD PUBLIC OperatorHome : E_RpcMethodResponse

VAR_INPUT requestId : ULINT; END_VAR
OperatorHome := _operatorMailbox.Submit(requestId := requestId, command := E_OperatorCommand.Home, value := 0.0);
END_METHOD

{attribute 'TcRpcEnable' := '1'}
METHOD PUBLIC OperatorPause : E_RpcMethodResponse

VAR_INPUT requestId : ULINT; END_VAR
OperatorPause := _operatorMailbox.Submit(requestId := requestId, command := E_OperatorCommand.Pause, value := 0.0);
END_METHOD

{attribute 'TcRpcEnable' := '1'}
METHOD PUBLIC OperatorProceed : E_RpcMethodResponse

VAR_INPUT requestId : ULINT; END_VAR
OperatorProceed := _operatorMailbox.Submit(requestId := requestId, command := E_OperatorCommand.Proceed, value := 0.0);
END_METHOD

{attribute 'TcRpcEnable' := '1'}
METHOD PUBLIC OperatorRetry : E_RpcMethodResponse

VAR_INPUT requestId : ULINT; END_VAR
OperatorRetry := _operatorMailbox.Submit(requestId := requestId, command := E_OperatorCommand.Retry, value := 0.0);
END_METHOD

{attribute 'TcRpcEnable' := '1'}
METHOD PUBLIC OperatorStart : E_RpcMethodResponse

VAR_INPUT requestId : ULINT; END_VAR
OperatorStart := _operatorMailbox.Submit(requestId := requestId, command := E_OperatorCommand.Start, value := 0.0);
END_METHOD

{attribute 'TcRpcEnable' := '1'}
METHOD PUBLIC OperatorStop : E_RpcMethodResponse

VAR_INPUT requestId : ULINT; END_VAR
OperatorStop := _operatorMailbox.Submit(requestId := requestId, command := E_OperatorCommand.Stop, value := 0.0);
END_METHOD

{attribute 'TcRpcEnable' := '1'}
METHOD PUBLIC OperatorReset : E_RpcMethodResponse
VAR_INPUT requestId : ULINT; END_VAR
OperatorReset := _operatorMailbox.Submit(requestId := requestId, command := E_OperatorCommand.Reset, value := 0.0);
END_METHOD

METHOD PUBLIC MapHomeCondition
VAR_INPUT
    bitIndex : UDINT;
    bGood : BOOL;
END_VAR
permHome.MapInput(bitIndex := bitIndex, inputValue := bGood);
END_METHOD

METHOD PUBLIC MapStartCondition
VAR_INPUT
    bitIndex : UDINT;
    bGood : BOOL;
END_VAR
permStart.MapInput(bitIndex := bitIndex, inputValue := bGood);
END_METHOD

METHOD PUBLIC MapProceedCondition
VAR_INPUT
    bitIndex : UDINT;
    bGood : BOOL;
END_VAR
permProceed.MapInput(bitIndex := bitIndex, inputValue := bGood);
END_METHOD

METHOD PUBLIC MapAutoCondition
VAR_INPUT
    bitIndex : UDINT;
    bGood : BOOL;
END_VAR
permAuto.MapInput(bitIndex := bitIndex, inputValue := bGood);
END_METHOD

METHOD INTERNAL ObserveStep
VAR_INPUT nStep : DINT; END_VAR
IF nStep = Status.Step.Current AND nStep MOD 2 = 0 AND Status.ActiveState THEN
    IF _activeStepCalls < 2 THEN _activeStepCalls := _activeStepCalls + 1; END_IF;
END_IF;
END_METHOD

METHOD INTERNAL CanExecuteStep : BOOL
VAR_INPUT nStep : DINT; END_VAR
CanExecuteStep := nStep = Status.Step.Current AND nStep MOD 2 = 0 AND
    _IsStepInStateRange(state := Status.State, nStep := nStep) AND
    NOT _stepFailurePending AND NOT Status.ShutdownFailed AND
    (NOT IsFaulted() OR Status.State = E_SM_State.STOPPING OR Status.State = E_SM_State.ABORTING);
END_METHOD

METHOD INTERNAL ValidateStep : BOOL
VAR_INPUT nStep : DINT; nDestination : DINT; nTimeout : DINT; END_VAR
ValidateStep := nTimeout >= 0 AND nTimeout <= 356400 AND (nDestination = 0 OR
    (_IsStepInStateRange(state := Status.State, nStep := nDestination) AND nDestination MOD 2 = 0 AND nDestination <> nStep));
IF NOT ValidateStep THEN
    _RaiseStepFault(stepNum := nStep, stepName := Status.Step.Name,
        code := E_SM_Fault.InvalidStepConfiguration, reason := 'Invalid timeout or destination; use zero or another even step in this state');
END_IF;
END_METHOD

METHOD PROTECTED _DispatchOperatorCommand : E_RpcMethodResponse
VAR_INPUT command : E_OperatorCommand; value : REAL; END_VAR
CASE command OF
E_OperatorCommand.Home: _DispatchOperatorCommand := THIS^.Home(eRequester := E_Requester.OPERATOR);
E_OperatorCommand.Start: _DispatchOperatorCommand := THIS^.Start(eRequester := E_Requester.OPERATOR);
E_OperatorCommand.Stop: _DispatchOperatorCommand := THIS^.Stop(eRequester := E_Requester.OPERATOR);
E_OperatorCommand.Abort: _DispatchOperatorCommand := THIS^.Abort(eRequester := E_Requester.OPERATOR);
E_OperatorCommand.Pause: _DispatchOperatorCommand := THIS^.Pause(eRequester := E_Requester.OPERATOR);
E_OperatorCommand.Proceed: _DispatchOperatorCommand := THIS^.Proceed(eRequester := E_Requester.OPERATOR);
E_OperatorCommand.Retry: _DispatchOperatorCommand := THIS^.Retry(eRequester := E_Requester.OPERATOR);
ELSE _DispatchOperatorCommand := SUPER^._DispatchOperatorCommand(command := command, value := value);
END_CASE;
END_METHOD

END_FUNCTION_BLOCK

// ---- POUs/Logic/Sequencing/StateMachine/FB_Step.TcPOU
(*
FB_Step - Lightweight step lifecycle wrapper
============================================
Each step in a sequence is one FB_Step instance. The parent FB_StateMachine
owns the active step number, step timer, fault detection, and command handling.
This FB only reports "am I active?" and drives the Entry/Execute/Exit/Advance
lifecycle for the user's code.

Lifecycle (while this step is the SM's active step):
  Entry   : TRUE one scan on activation         -> one-shot init
  Execute : TRUE every scan until perms satisfied -> cyclic work + MapPerm
  Exiting : TRUE one scan after perms satisfied  -> one-shot cleanup
  Advance : writes nNextStep to the SM, SM increments on next scan

Branching / looping / jumping:
  nNextStep is a VAR_INPUT re-evaluated every scan. To branch, loop, or jump,
  just assign nNextStep dynamically in the call. There is no separate override
  method -- the input IS the dynamic target.

      step(sm := sm, nStep := 3004,
           nNextStep := SEL(bPass, 3500, 3006),  // branch inline
           nTimeout := 12, sName := 'Inspect');

  nNextStep := 0   -> completes the sequence (SM transitions to waiting state)
  nNextStep := N   -> SM advances to step N (any valid step; forward/back)

Note: 'Exiting' is used instead of 'Exit' because EXIT is an IEC reserved word.
*)
FUNCTION_BLOCK FB_Step
VAR_IN_OUT
sm : FB_StateMachine;
END_VAR

VAR_INPUT
    nRequired : ULINT;
    // Required completion conditions, declared independently of MapPerm calls.
    nStep : DINT;
    nNextStep : DINT;
    nTimeout : DINT;
    sName : STRING(40);
END_VAR

VAR_OUTPUT
    Entry : BOOL;
    Execute : BOOL;
    Exiting : BOOL;
END_VAR

VAR
    _perms : FB_Permissives;
    _active : BOOL;
    _prevActive : BOOL;
    _permsSatisfied : BOOL;
    _permsEvalReady : BOOL;
    _exitDone : BOOL;
END_VAR

// Evaluate independently declared required completion conditions.
_perms.cfg.nRequired := nRequired;
_perms();
_permsSatisfied := _perms.sts.bOK;

// Every called instance contributes to the parent's previous-scan coverage check.
sm.ObserveStep(nStep := nStep);
_active := sm.CanExecuteStep(nStep := nStep);
IF _active THEN
    _active := sm.ValidateStep(nStep := nStep, nDestination := nNextStep, nTimeout := nTimeout);
END_IF;

// Reset lifecycle outputs each scan
Entry := FALSE;
Execute := FALSE;
Exiting := FALSE;

// Timeout applies to the entire active lifecycle, including Entry and Exiting.
IF _active AND nTimeout > 0 AND sm.Status.Step.TimerSeconds >= DINT_TO_REAL(nTimeout) THEN
    sm._RaiseStepFault(stepNum := nStep, stepName := sName, code := E_SM_Fault.StepTimeout, reason := '');
    _active := FALSE;
END_IF;

IF _active THEN
    // Publish step name to SM for HMI / diagnostics
    sm.SetStepName(sName);
    sm.SetStepPermissives(cfg := _perms.cfg, sts := _perms.sts);

    IF NOT _prevActive THEN
        //---------------------------------------------------------------------
        // ENTRY: first scan this step is active
        //---------------------------------------------------------------------
        Entry := TRUE;
        _permsEvalReady := FALSE;
        _exitDone := FALSE;

    ELSIF NOT _permsEvalReady THEN
        //---------------------------------------------------------------------
        // First EXECUTE scan: user is mapping perms this scan; evaluate next
        // scan so the first evaluation sees all MapPerm calls from this cycle.
        //---------------------------------------------------------------------
        Execute := TRUE;
        _permsEvalReady := TRUE;

    ELSIF NOT _permsSatisfied THEN
        //---------------------------------------------------------------------
        // EXECUTE: waiting for all mapped permissives to be satisfied
        //---------------------------------------------------------------------
        IF NOT sm.IsFaulted() OR sm.Status.State = E_SM_State.ABORTING OR sm.Status.State = E_SM_State.STOPPING THEN
            Execute := TRUE;
        END_IF;

    ELSIF NOT _exitDone THEN
        //---------------------------------------------------------------------
        // EXIT: all permissives satisfied, one-scan cleanup
        //---------------------------------------------------------------------
        Exiting := TRUE;
        _exitDone := TRUE;

    ELSE
        //---------------------------------------------------------------------
        // ADVANCE: post-exit, hand the (current-scan) nNextStep to the SM.
        // Because nNextStep is re-evaluated every scan, the user's latest
        // branch decision wins -- no override method needed.
        //---------------------------------------------------------------------
        sm.SetNextStep(nStep := nNextStep);
    END_IF;

ELSE
    // Reset lifecycle tracking when step is not active
    _permsEvalReady := FALSE;
    _exitDone := FALSE;
END_IF;

_prevActive := _active;

METHOD MapPerm
VAR_INPUT
    nIndex : UDINT;
    sDescription : STRING;
    bValue : BOOL;
END_VAR
IF nIndex > 63 THEN
    RETURN;
END_IF;
_perms.MapInput(bitIndex := nIndex, inputValue := bValue);
_perms.cfg.aNames[nIndex] := sDescription;
END_METHOD

// Record a fault from an active step; nonpositive codes normalize to StepUserFault.
// Ordinary work lands on its odd recovery step. Failed Stop escalates to Abort;
// failed Abort latches ShutdownFailed and enters STOPPED on the next SM call.
// Lifecycle outputs are cleared immediately. Call only after FB_Step(sm := ...).
// Subsequent calls are ignored until the step is explicitly reactivated.
//
// C0371 is the "VAR_IN_OUT accessed from method" warning. Safe here because
// RaiseFault is only legal inside a step block, after FB_Step() has been
// called with a valid sm reference.
METHOD RaiseFault
VAR_INPUT
    code   : DINT;
    reason : STRING(79);
END_VAR
{warning disable C0371}
IF NOT _active THEN
    RETURN;
END_IF;

sm._RaiseStepFault(
stepNum  := nStep,
stepName := sName,
code     := code,
reason   := reason
);
Entry := FALSE;
Execute := FALSE;
Exiting := FALSE;
_active := FALSE;
{warning restore C0371}
END_METHOD

END_FUNCTION_BLOCK

// ---- POUs/IO/DigitalInput/FB_DigitalInput.TcPOU
// Generic digital input conditioner.
//
// Pipeline:
//   terminal bit (inSignal) -> quality gate -> invert -> asymmetric
//   debounce -> edge detection -> sts.value / risingEdge / fallingEdge
//
// Quality handling: while inpQuality is BAD the raw reading is ignored and
// the previous rawValue is held. If the input stays BAD longer than
// cfg.qualityFaultAfter the FB raises E_DigitalInput_Fault.BadQuality
// through the fault book-keeping inherited from FB_DeviceBase.
//
// Debounce is asymmetric on purpose: many sensors need a short ON-delay to
// reject noise but should drop out instantly when they go dark (or vice
// versa). Setting both times to T#0MS disables the filter.
{attribute 'OPC.UA.DA' := '1'}
FUNCTION_BLOCK FB_DigitalInput EXTENDS FB_DeviceBase
VAR_INPUT
    {attribute 'OPC.UA.DA' := '0'}
    inSignal : BOOL;
    {attribute 'OPC.UA.DA' := '1'}
    {attribute 'OPC.UA.DA.Access' := '1'}
    cfg        : ST_DigitalInput_Cfg;
    {attribute 'OPC.UA.DA' := '0'}
    inpQuality : E_IO_Quality := E_IO_Quality.GOOD;
END_VAR

VAR_OUTPUT
    {attribute 'OPC.UA.DA' := '1'}
    {attribute 'OPC.UA.DA.Access' := '1'}
    sts : ST_DigitalInput_Sts;
END_VAR

VAR

    // Debounce timers (asymmetric ON / OFF delays).
    {attribute 'OPC.UA.DA' := '0'}
    _tonOn          : TON;
    {attribute 'OPC.UA.DA' := '0'}
    _tofOff         : TON;
    _conditioningKnown : BOOL;
    _previousCfg : ST_DigitalInput_Cfg;
    _conditioningChanged : BOOL;

    // Quality watchdog — ticks for every unusable quality value.
    {attribute 'OPC.UA.DA' := '0'}
    _tonBadQuality  : TON;

    // Scratch values.
    {attribute 'OPC.UA.DA' := '0'}
    _rawBool        : BOOL;
    {attribute 'OPC.UA.DA' := '0'}
    _invertedBool   : BOOL;
    {attribute 'OPC.UA.DA' := '0'}
    _debouncedBool  : BOOL;
    {attribute 'OPC.UA.DA' := '0'}
    _prevDebounced  : BOOL;
END_VAR

_ProcessOperatorCommands();
// Configuration changes cannot borrow elapsed evidence from the previous interpretation.
_conditioningChanged := _conditioningKnown AND (cfg.invert <> _previousCfg.invert OR
    cfg.debounceOn <> _previousCfg.debounceOn OR cfg.debounceOff <> _previousCfg.debounceOff);
_previousCfg := cfg; _conditioningKnown := TRUE;
IF _conditioningChanged THEN _tonOn(IN := FALSE); _tofOff(IN := FALSE); END_IF;
sts.quality := inpQuality;
sts.risingEdge := FALSE; sts.fallingEdge := FALSE;
IF inpQuality = E_IO_Quality.GOOD OR inpQuality = E_IO_Quality.CLAMPED THEN
    _rawBool := inSignal;
    _invertedBool := _rawBool XOR cfg.invert;
    // Time each transition from fresh evidence, holding the established state meanwhile.
    IF _invertedBool THEN
        _tofOff(IN := FALSE);
        IF NOT _debouncedBool THEN
            _tonOn(IN := TRUE, PT := cfg.debounceOn);
            IF _tonOn.Q THEN _debouncedBool := TRUE; END_IF;
        ELSE _tonOn(IN := FALSE); END_IF;
    ELSE
        _tonOn(IN := FALSE);
        IF _debouncedBool THEN
            _tofOff(IN := TRUE, PT := cfg.debounceOff);
            IF _tofOff.Q THEN _debouncedBool := FALSE; END_IF;
        ELSE _tofOff(IN := FALSE); END_IF;
    END_IF;
    sts.risingEdge := _debouncedBool AND NOT _prevDebounced;
    sts.fallingEdge := NOT _debouncedBool AND _prevDebounced;
    _prevDebounced := _debouncedBool;
    sts.value := _debouncedBool;
    sts.rawValue := _rawBool;
ELSE
    // Invalid elapsed time is not debounce evidence. Keep published value/raw unchanged.
    _tonOn(IN := FALSE); _tofOff(IN := FALSE);
END_IF;

// 6. Quality watchdog. Enabled only when qualityFaultAfter > 0.
_tonBadQuality(
    IN := NOT (inpQuality = E_IO_Quality.GOOD OR inpQuality = E_IO_Quality.CLAMPED) AND cfg.qualityFaultAfter > T#0MS,
    PT := cfg.qualityFaultAfter
);

IF _tonBadQuality.Q THEN
    _Raise(
        code   := E_DigitalInput_Fault.BadQuality,
        source := 'QUALITY',
        reason := 'inpQuality stayed unusable past qualityFaultAfter'
    );
END_IF;

// 7. Refresh shared header (fault surface, ready flags, timestamps).
_UpdateHeader(header := sts.header, stateString := '', busy := FALSE);

// Maps E_DigitalInput_Fault codes to human-readable strings for the HMI.
METHOD PROTECTED ResolveFaultString : STRING(79)
VAR_INPUT
    code : DINT;
END_VAR
CASE code OF
    0:
        ResolveFaultString := '';
    E_DigitalInput_Fault.BadQuality:
        ResolveFaultString := 'Signal quality BAD past configured timeout';
    E_DigitalInput_Fault.StuckHigh:
        ResolveFaultString := 'Debounced signal stuck HIGH past configured timeout';
    E_DigitalInput_Fault.StuckLow:
        ResolveFaultString := 'Debounced signal stuck LOW past configured timeout';
ELSE
    ResolveFaultString := CONCAT('DigitalInput fault ', DINT_TO_STRING(code));
END_CASE;
END_METHOD

// Owning-task application API: invalidate history before binding a different source.
METHOD PUBLIC ReassignInput
_tonOn(IN := FALSE); _tofOff(IN := FALSE); _tonBadQuality(IN := FALSE);
_debouncedBool := FALSE; _prevDebounced := FALSE; _rawBool := FALSE;
sts.value := FALSE; sts.rawValue := FALSE;
sts.risingEdge := FALSE; sts.fallingEdge := FALSE;
sts.quality := E_IO_Quality.UNKNOWN;
_conditioningKnown := FALSE;
END_METHOD

END_FUNCTION_BLOCK

// ---- POUs/IO/DigitalOutput/FB_DigitalOutput.TcPOU
// Generic digital output driver.
//
// Pipeline:
//   SetOn / SetOff -> explicit request -> quality gate -> asymmetric
//   debounce -> mode (Regular | SinglePulse | ContinuousPulse) -> invert
//   (Regular only) -> terminal bit (outSignal)
//
// Saved intent is restored only with cfg.restoreCommandOnRestart.
// Quality loss disarms output; recovery requires a fresh accepted command.
// ForceSafe and Reset inhibit output independent of the previous command.
//
// Inversion deliberately only applies in Regular mode — inverting a pulse
// train just phase-shifts it, which is rarely what the author means. Pulse
// behaviour should be shaped through cfg.pulseOn / cfg.pulseOff.
{attribute 'OPC.UA.DA' := '1'}
FUNCTION_BLOCK FB_DigitalOutput EXTENDS FB_DeviceBase
VAR_INPUT
    {attribute 'OPC.UA.DA' := '1'}
    {attribute 'OPC.UA.DA.Access' := '1'}
    cfg        : ST_DigitalOutput_Cfg;
    {attribute 'OPC.UA.DA' := '0'}
    inpQuality : E_IO_Quality := E_IO_Quality.GOOD;
END_VAR

VAR_OUTPUT
    {attribute 'OPC.UA.DA' := '1'}
    {attribute 'OPC.UA.DA.Access' := '1'}
    outSignal : BOOL;
    {attribute 'OPC.UA.DA' := '1'}
    {attribute 'OPC.UA.DA.Access' := '1'}
    sts : ST_DigitalOutput_Sts;
END_VAR

VAR PERSISTENT
    // Saved intent and validity; durability depends on target persistent saving.
    {attribute 'OPC.UA.DA' := '0'}
    _savedCommand : BOOL;
    {attribute 'OPC.UA.DA' := '0'}
    _savedCommandValid : BOOL;
END_VAR

VAR
    _configurationKnown : BOOL;
    _lastConfiguration : ST_DigitalOutput_Cfg;
    _requestSync : BOOL; // Operating intent is never restored implicitly.
    _armed : BOOL;
    _commandReceived : BOOL;
    _startup : BOOL := TRUE;
    _forceSafe : BOOL;
    _safeRequested : BOOL;
    _qualityGood : BOOL;

    // Debounce of commanded value.
    {attribute 'OPC.UA.DA' := '0'}
    _tonOn          : TON;
    {attribute 'OPC.UA.DA' := '0'}
    _tofOff         : TOF;

    // Pulse-mode timers.
    {attribute 'OPC.UA.DA' := '0'}
    _tonPulseOn     : TON;
    {attribute 'OPC.UA.DA' := '0'}
    _tonPulseOff    : TON;

    // Quality watchdog.
    {attribute 'OPC.UA.DA' := '0'}
    _tonBadQuality  : TON;

    // Scratch state.
    {attribute 'OPC.UA.DA' := '0'}
    _debouncedCmd   : BOOL;
    {attribute 'OPC.UA.DA' := '0'}
    _prevDebounced  : BOOL;
    {attribute 'OPC.UA.DA' := '0'}
    _pulseActive    : BOOL;
    {attribute 'OPC.UA.DA' := '0'}
    _finalOutput    : BOOL;
    {attribute 'OPC.UA.DA' := '0'}
    _prevPhysical   : BOOL;
END_VAR

_SyncConfiguration();
_ProcessOperatorCommands();
_qualityGood := inpQuality = E_IO_Quality.GOOD OR inpQuality = E_IO_Quality.CLAMPED;
IF _startup THEN
    _startup := FALSE;
    // A valid marker in a missing/backup image cannot authorize old operating intent.
    // A command accepted in this execution is fresh and does not depend on that image.
    IF NOT _commandReceived AND NOT THIS^._HasTrustedPersistentImage() THEN
        _savedCommandValid := FALSE;
    END_IF;
    IF NOT _commandReceived AND cfg.restoreCommandOnRestart AND _savedCommandValid THEN
        _requestSync := _savedCommand;
        _armed := TRUE;
    END_IF;
END_IF;
IF NOT _qualityGood THEN _armed := FALSE; END_IF;
// 1. Publish quality + commanded value before any gating.
sts.quality   := inpQuality;
sts.commanded := _requestSync;

// 2. Asymmetric debounce on commanded value. Keeps pulse timers in sync
//    with the debounced edge, not the raw request.
_tonOn (IN := _requestSync, PT := cfg.debounceOn);
_tofOff(IN := _requestSync, PT := cfg.debounceOff);

IF _requestSync AND _tonOn.Q THEN
    _debouncedCmd := TRUE;
ELSIF NOT _requestSync AND NOT _tofOff.Q THEN
    _debouncedCmd := FALSE;
END_IF;

// 3. Mode shaping.
CASE cfg.mode OF
    E_DigitalOutput_Mode.Regular:
        _tonPulseOn (IN := FALSE);
        _tonPulseOff(IN := FALSE);
        _pulseActive := FALSE;
        IF cfg.invert THEN
            _finalOutput := NOT _debouncedCmd;
        ELSE
            _finalOutput := _debouncedCmd;
        END_IF;

    E_DigitalOutput_Mode.SinglePulse:
        // Rising edge of debounced command arms the one-shot.
        IF _debouncedCmd AND NOT _prevDebounced THEN
            _pulseActive := TRUE;
            _tonPulseOn(IN := FALSE);
        END_IF;

        IF _pulseActive THEN
            _tonPulseOn(IN := TRUE, PT := cfg.pulseOn);
            IF _tonPulseOn.Q THEN
                _pulseActive := FALSE;
            END_IF;
        END_IF;

        // Commanded-LOW disarms the pulse early so operators can cancel.
        IF NOT _debouncedCmd THEN
            _pulseActive := FALSE;
            _tonPulseOn(IN := FALSE);
        END_IF;

        _tonPulseOff(IN := FALSE);
        _finalOutput := _pulseActive AND NOT _tonPulseOn.Q;

    E_DigitalOutput_Mode.ContinuousPulse:
        // While the command is TRUE, alternate ON / OFF using the two
        // pulse timers as a simple state machine.
        IF _debouncedCmd THEN
            IF _pulseActive THEN
                _tonPulseOn (IN := TRUE, PT := cfg.pulseOn);
                _tonPulseOff(IN := FALSE);
                IF _tonPulseOn.Q THEN
                    _pulseActive := FALSE;
                    _tonPulseOn(IN := FALSE);
                END_IF;
            ELSE
                _tonPulseOff(IN := TRUE, PT := cfg.pulseOff);
                _tonPulseOn (IN := FALSE);
                IF _tonPulseOff.Q THEN
                    _pulseActive := TRUE;
                    _tonPulseOff(IN := FALSE);
                END_IF;
            END_IF;
            _finalOutput := _pulseActive;
        ELSE
            _pulseActive := FALSE;
            _tonPulseOn (IN := FALSE);
            _tonPulseOff(IN := FALSE);
            _finalOutput := FALSE;
        END_IF;
ELSE
    _finalOutput := cfg.safeOutput;
    _armed := FALSE;
END_CASE;

// 6. Quality watchdog.
_tonBadQuality(
    IN := NOT _qualityGood AND cfg.qualityFaultAfter > T#0MS,
    PT := cfg.qualityFaultAfter
);

IF _tonBadQuality.Q THEN
    _Raise(
        code   := E_DigitalOutput_Fault.BadQuality,
        source := 'QUALITY',
        reason := 'inpQuality stayed BAD past qualityFaultAfter'
    );
END_IF;


IF NOT (cfg.mode = E_DigitalOutput_Mode.Regular OR cfg.mode = E_DigitalOutput_Mode.SinglePulse OR cfg.mode = E_DigitalOutput_Mode.ContinuousPulse) OR
   (cfg.mode <> E_DigitalOutput_Mode.Regular AND cfg.pulseOn = T#0MS) OR
   (cfg.mode = E_DigitalOutput_Mode.ContinuousPulse AND cfg.pulseOff = T#0MS) THEN
    _Raise(code := E_DigitalOutput_Fault.BadConfig, source := 'CONFIG', reason := 'Invalid output mode or pulse duration');
END_IF;
IF IsFaulted() THEN _armed := FALSE; END_IF;
// Final output policy. Bad quality disarms; returning quality cannot restart output.
IF _forceSafe OR IsFaulted() OR (_qualityGood AND NOT _armed) THEN
    outSignal := cfg.safeOutput;
ELSIF NOT _qualityGood THEN
    IF NOT cfg.holdOnBadQuality THEN outSignal := cfg.safeOutput; END_IF;
ELSE
    outSignal := _finalOutput;
END_IF;
IF NOT _armed OR _forceSafe THEN
    _tonOn(IN := FALSE); _tofOff(IN := FALSE);
    _tonPulseOn(IN := FALSE); _tonPulseOff(IN := FALSE);
    _debouncedCmd := FALSE; _pulseActive := FALSE;
END_IF;

// 5. Edge pulses reflect the *physical* output, not the command.
sts.risingEdge  :=      outSignal AND NOT _prevPhysical;
sts.fallingEdge := NOT outSignal AND     _prevPhysical;
_prevPhysical := outSignal;
_prevDebounced := _debouncedCmd;

sts.value := outSignal;
sts.outputInhibited := NOT _armed OR _forceSafe OR IsFaulted();

_safeRequested := FALSE; // consumed after applying outputs

// 7. Refresh shared header.
_UpdateHeader(header := sts.header, stateString := '', busy := FALSE);

METHOD PUBLIC SetOn : E_RpcMethodResponse
VAR_INPUT
    eRequester : E_Requester := E_Requester.PROG;
END_VAR
// Reject invalid identity before any command-specific mutation.
SetOn := F_ValidateRequester(eRequester := eRequester, bSourceLocked := FALSE, bFaulted := FALSE);
IF SetOn <> E_RpcMethodResponse.ACCEPTED THEN RETURN; END_IF;
_SyncConfiguration();
IF _safeRequested THEN
    SetOn := E_RpcMethodResponse.REJECTED_INTERLOCKED;
    RETURN;
END_IF;
SetOn := F_ValidateRequester(
    eRequester    := eRequester,
    bSourceLocked := bSourceLockedToProg,
    bFaulted      := IsFaulted()
);

IF SetOn <> E_RpcMethodResponse.ACCEPTED THEN
    RETURN;
END_IF;

_requestSync := TRUE;
_savedCommand := _requestSync;
_savedCommandValid := TRUE;
_armed := TRUE;
_commandReceived := TRUE;
_forceSafe := FALSE;
_AcceptCommand(eRequester := eRequester);
END_METHOD

METHOD PUBLIC SetOff : E_RpcMethodResponse
VAR_INPUT
    eRequester : E_Requester := E_Requester.PROG;
END_VAR
// Reject invalid identity before any command-specific mutation.
SetOff := F_ValidateRequester(eRequester := eRequester, bSourceLocked := FALSE, bFaulted := FALSE);
IF SetOff <> E_RpcMethodResponse.ACCEPTED THEN RETURN; END_IF;
_SyncConfiguration();
IF _safeRequested THEN
    SetOff := E_RpcMethodResponse.REJECTED_INTERLOCKED;
    RETURN;
END_IF;
_operatorMailbox.CancelNormal();
_requestSync := FALSE;
_savedCommand := FALSE;
_savedCommandValid := TRUE;
_armed := TRUE;
_commandReceived := TRUE;
_forceSafe := FALSE;
_AcceptCommand(eRequester := eRequester);
SetOff := E_RpcMethodResponse.ACCEPTED;
END_METHOD

METHOD PROTECTED ResolveFaultString : STRING(79)
VAR_INPUT
    code : DINT;
END_VAR
CASE code OF
    E_DigitalOutput_Fault.BadConfig: ResolveFaultString := 'Digital output configuration invalid';
    0:
        ResolveFaultString := '';
    E_DigitalOutput_Fault.BadQuality:
        ResolveFaultString := 'Output quality BAD past configured timeout';
ELSE
    ResolveFaultString := CONCAT('DigitalOutput fault ', DINT_TO_STRING(code));
END_CASE;
END_METHOD

{attribute 'TcRpcEnable' := '1'}
METHOD PUBLIC OperatorSetOn : E_RpcMethodResponse

VAR_INPUT requestId : ULINT; END_VAR
OperatorSetOn := _operatorMailbox.Submit(requestId := requestId, command := E_OperatorCommand.SetOn, value := 0.0);
END_METHOD

{attribute 'TcRpcEnable' := '1'}
METHOD PUBLIC OperatorSetOff : E_RpcMethodResponse

VAR_INPUT requestId : ULINT; END_VAR
OperatorSetOff := _operatorMailbox.Submit(requestId := requestId, command := E_OperatorCommand.SetOff, value := 0.0);
END_METHOD

METHOD PUBLIC ForceSafe : E_RpcMethodResponse
VAR_INPUT
    eRequester : E_Requester := E_Requester.PROG;
END_VAR
// Reject invalid identity before any command-specific mutation.
ForceSafe := F_ValidateRequester(eRequester := eRequester, bSourceLocked := FALSE, bFaulted := FALSE);
IF ForceSafe <> E_RpcMethodResponse.ACCEPTED THEN RETURN; END_IF;
_SyncConfiguration();
_operatorMailbox.CancelNormal();
_safeRequested := TRUE;
_armed := FALSE;
_forceSafe := TRUE;
_requestSync := FALSE;
_savedCommand := _requestSync;
_savedCommandValid := FALSE;
_AcceptCommand(eRequester := eRequester);
ForceSafe := E_RpcMethodResponse.ACCEPTED;
END_METHOD

{attribute 'TcRpcEnable' := '1'}
METHOD PUBLIC OperatorForceSafe : E_RpcMethodResponse
VAR_INPUT requestId : ULINT; END_VAR
OperatorForceSafe := _operatorMailbox.Submit(requestId := requestId, command := E_OperatorCommand.ForceSafe, value := 0.0);
END_METHOD

METHOD PUBLIC Reset : E_RpcMethodResponse
VAR_INPUT
    eRequester : E_Requester := E_Requester.PROG;
END_VAR
// Reject invalid identity before any command-specific mutation.
Reset := F_ValidateRequester(eRequester := eRequester, bSourceLocked := FALSE, bFaulted := FALSE);
IF Reset <> E_RpcMethodResponse.ACCEPTED THEN RETURN; END_IF;
_SyncConfiguration();
_operatorMailbox.CancelNormal();
ForceSafe(eRequester := eRequester);
Reset := SUPER^.Reset(eRequester := eRequester);
END_METHOD

METHOD PROTECTED _DispatchOperatorCommand : E_RpcMethodResponse
VAR_INPUT command : E_OperatorCommand; value : REAL; END_VAR
CASE command OF
E_OperatorCommand.SetOn: _DispatchOperatorCommand := THIS^.SetOn(eRequester := E_Requester.OPERATOR);
E_OperatorCommand.SetOff: _DispatchOperatorCommand := THIS^.SetOff(eRequester := E_Requester.OPERATOR);
E_OperatorCommand.ForceSafe: _DispatchOperatorCommand := THIS^.ForceSafe(eRequester := E_Requester.OPERATOR);
ELSE _DispatchOperatorCommand := SUPER^._DispatchOperatorCommand(command := command, value := value);
END_CASE;
END_METHOD

METHOD PRIVATE _SyncConfiguration
// Configuration is owned by the same cyclic task as this device.
// The first observation establishes a baseline and preserves first-scan commands.
IF NOT _configurationKnown THEN
    _lastConfiguration := cfg;
    _configurationKnown := TRUE;
    RETURN;
END_IF;
IF cfg.restoreCommandOnRestart <> _lastConfiguration.restoreCommandOnRestart OR
   cfg.holdOnBadQuality <> _lastConfiguration.holdOnBadQuality OR
   cfg.safeOutput <> _lastConfiguration.safeOutput OR
   cfg.invert <> _lastConfiguration.invert OR
   cfg.debounceOn <> _lastConfiguration.debounceOn OR
   cfg.debounceOff <> _lastConfiguration.debounceOff OR
   cfg.mode <> _lastConfiguration.mode OR
   cfg.pulseOn <> _lastConfiguration.pulseOn OR
   cfg.pulseOff <> _lastConfiguration.pulseOff OR
   cfg.qualityFaultAfter <> _lastConfiguration.qualityFaultAfter THEN
    // Discard old operating intent before interpreting it under a new configuration.
    _operatorMailbox.CancelNormal(includeSetOff := TRUE);
    _armed := FALSE;
    _forceSafe := TRUE;
    _requestSync := FALSE;
    _savedCommand := FALSE;
    _savedCommandValid := FALSE;
    _commandReceived := TRUE;
    _tonOn(IN := FALSE);
    _tofOff(IN := FALSE, PT := T#0MS);
    _tonPulseOn(IN := FALSE);
    _tonPulseOff(IN := FALSE);
    _tonBadQuality(IN := FALSE);
    _debouncedCmd := FALSE;
    _prevDebounced := FALSE;
    _pulseActive := FALSE;
END_IF;
_lastConfiguration := cfg;
END_METHOD

// Runtime provenance gate, overridable by policy-test probes without system writes.
// A successful load does not establish that the latest command was durably saved.
METHOD PROTECTED _HasTrustedPersistentImage : BOOL
_HasTrustedPersistentImage := TwinCAT_SystemInfoVarList._AppInfo.BootDataLoaded
    AND NOT TwinCAT_SystemInfoVarList._AppInfo.OldBootData;
END_METHOD

END_FUNCTION_BLOCK

// ---- POUs/IO/AnalogInput/FB_AnalogInput.TcPOU
// Generic analog input conditioner.
//
// Pipeline:
//   UNION terminal -> type select -> quality gate -> clamp to scaling range
//   -> linear EU scaling -> optional first-order LPF -> sts
//
// The UNION input (inRaw) means one FB instance handles any raw form the
// hardware produces â€” 0-10 V (INT), 4-20 mA (INT), 32-bit counter (UDINT),
// scaled REAL, bit-packed WORD, etc. Pick the interpretation with
// cfg.inputType.
//
// Scope: conditioning only. Process-alarm limits (HH / HI / LO / LL),
// latching, severity, and ack all live on FB_AlarmLimit â€” compose it with
// sts.value if you need that behaviour. Faults here are restricted to
// ground truths about the signal itself (quality, clamp, bad config).
{attribute 'OPC.UA.DA' := '1'}
FUNCTION_BLOCK FB_AnalogInput EXTENDS FB_DeviceBase
VAR_INPUT
    {attribute 'OPC.UA.DA' := '0'}
    inRaw : U_IoRaw_In;
    {attribute 'OPC.UA.DA' := '1'}
    {attribute 'OPC.UA.DA.Access' := '1'}
    cfg        : ST_AnalogInput_Cfg;
    {attribute 'OPC.UA.DA' := '0'}
    inpQuality : E_IO_Quality := E_IO_Quality.GOOD;
END_VAR

VAR_OUTPUT
    {attribute 'OPC.UA.DA' := '1'}
    {attribute 'OPC.UA.DA.Access' := '1'}
    sts : ST_AnalogInput_Sts;
END_VAR

VAR
    _inputSnapshot : U_IoRaw_In;
    _lastConditioningCfg : ST_AnalogInput_Cfg;
    _conditioningCfgKnown : BOOL;
    _hasValidSample : BOOL;
    _reseedPending : BOOL;

    // Commissioning state.
    {attribute 'OPC.UA.DA' := '0'}
    _firstScan     : BOOL := TRUE;
    {attribute 'OPC.UA.DA' := '0'}
    _configBad     : BOOL;
    {attribute 'OPC.UA.DA' := '0'}
    _taskDtSec     : REAL;

    // Filter + watchdog timers.
    {attribute 'OPC.UA.DA' := '0'}
    _filter        : FB_LPF_FirstOrder_IIR;
    {attribute 'OPC.UA.DA' := '0'}
    _tonBadQuality : TON;

    // Scratch values (reset every scan).
    {attribute 'OPC.UA.DA' := '0'}
    _rawReal       : REAL;
    _scaledWide    : LREAL;
    _signalBad     : BOOL;
    {attribute 'OPC.UA.DA' := '0'}
    _clampedRaw    : REAL;
    {attribute 'OPC.UA.DA' := '0'}
    _scaledReal    : REAL;
    {attribute 'OPC.UA.DA' := '0'}
    _finalReal     : REAL;
END_VAR

_ProcessOperatorCommands();
// 1. First scan: config validation + task dt cache for the filter.
IF _firstScan THEN
    _firstScan := FALSE;
    _taskDtSec := TIME_TO_REAL(F_GetTaskCycleTime()) / 1000.0;

END_IF;

// Classify representations before comparisons; NaN comparisons can stop the PLC.
_configBad := NOT F_IsFiniteReal(value := cfg.euMin) OR NOT F_IsFiniteReal(value := cfg.euMax) OR
              NOT F_IsFiniteReal(value := cfg.rawMin) OR NOT F_IsFiniteReal(value := cfg.rawMax);
IF NOT _configBad THEN
    _configBad := NOT cfg.useRawValue AND (cfg.rawMin >= cfg.rawMax OR cfg.euMin >= cfg.euMax);
END_IF;
_configBad := _configBad OR NOT (
    cfg.inputType = __SYSTEM.TYPE_CLASS.TYPE_INT OR cfg.inputType = __SYSTEM.TYPE_CLASS.TYPE_UINT OR
    cfg.inputType = __SYSTEM.TYPE_CLASS.TYPE_WORD OR cfg.inputType = __SYSTEM.TYPE_CLASS.TYPE_DINT OR
    cfg.inputType = __SYSTEM.TYPE_CLASS.TYPE_UDINT OR cfg.inputType = __SYSTEM.TYPE_CLASS.TYPE_DWORD OR
    cfg.inputType = __SYSTEM.TYPE_CLASS.TYPE_REAL);

// Only compare validated configurations; previous snapshots contain finite values.
IF NOT _configBad THEN
    IF _conditioningCfgKnown AND _hasValidSample THEN
        IF cfg.inputType <> _lastConditioningCfg.inputType OR
           cfg.useRawValue <> _lastConditioningCfg.useRawValue OR
           cfg.rawMin <> _lastConditioningCfg.rawMin OR cfg.rawMax <> _lastConditioningCfg.rawMax OR
           cfg.euMin <> _lastConditioningCfg.euMin OR cfg.euMax <> _lastConditioningCfg.euMax OR
           ((cfg.filterTau = T#0MS) <> (_lastConditioningCfg.filterTau = T#0MS)) THEN
            _reseedPending := TRUE;
        END_IF;
    END_IF;
    _lastConditioningCfg := cfg;
    _conditioningCfgKnown := TRUE;
END_IF;

sts.unit    := cfg.unit;
sts.quality := inpQuality;

// 2. Snapshot the selected source.
_inputSnapshot := inRaw;
CASE cfg.inputType OF
    __SYSTEM.TYPE_CLASS.TYPE_INT:   _rawReal := TO_REAL(_inputSnapshot.nInt);
    __SYSTEM.TYPE_CLASS.TYPE_UINT:  _rawReal := TO_REAL(_inputSnapshot.ui);
    __SYSTEM.TYPE_CLASS.TYPE_WORD:  _rawReal := TO_REAL(_inputSnapshot.w);
    __SYSTEM.TYPE_CLASS.TYPE_DINT:  _rawReal := TO_REAL(_inputSnapshot.di);
    __SYSTEM.TYPE_CLASS.TYPE_UDINT: _rawReal := TO_REAL(_inputSnapshot.udi);
    __SYSTEM.TYPE_CLASS.TYPE_DWORD: _rawReal := TO_REAL(_inputSnapshot.dw);
    __SYSTEM.TYPE_CLASS.TYPE_REAL:
    _rawReal := _inputSnapshot.fReal;
ELSE
    _rawReal := sts.rawReal;
END_CASE;

// 3. Quality-gated hold. Ignore the freshly read value while BAD.
_signalBad := NOT F_IsFiniteReal(value := _rawReal);
IF _signalBad OR _configBad THEN sts.quality := E_IO_Quality.BAD; END_IF;
IF _signalBad OR _configBad OR NOT (inpQuality = E_IO_Quality.GOOD OR inpQuality = E_IO_Quality.CLAMPED) THEN
    _rawReal := sts.rawReal;
END_IF;

sts.rawReal := _rawReal;

// Unusable samples cannot advance conditioning state or reinterpret held raw data.
// Preserve the last published value and filter history until a valid sample arrives.
_finalReal := sts.value;
IF NOT _configBad AND NOT _signalBad AND
   (inpQuality = E_IO_Quality.GOOD OR inpQuality = E_IO_Quality.CLAMPED) THEN
// 4. Raw-value bypass â€” no clamp / scale / filter.
IF cfg.useRawValue THEN
    _finalReal         := _rawReal;
    sts.scaled      := _rawReal;
    sts.clampedLow  := FALSE;
    sts.clampedHigh := FALSE;
    sts.clampActive := FALSE;
ELSE
    // 4a. Clamp-and-report against the scaling range. The same comparison
    //     drives both the scaling clamp and the sts.clamped* booleans so the
    //     HMI surface always matches what the math actually used.
    sts.clampedLow  := _rawReal < cfg.rawMin;
    sts.clampedHigh := _rawReal > cfg.rawMax;
    sts.clampActive := sts.clampedLow OR sts.clampedHigh;

    _clampedRaw := _rawReal;
    IF sts.clampedLow THEN
        _clampedRaw := cfg.rawMin;
    ELSIF sts.clampedHigh THEN
        _clampedRaw := cfg.rawMax;
    END_IF;

    // Promote quality tag while clamped (even if no fault is raised).
    IF sts.clampActive AND sts.quality = E_IO_Quality.GOOD THEN
        sts.quality := E_IO_Quality.CLAMPED;
    END_IF;

    // Wide intermediate math avoids overflow before range checks can act.
    IF NOT _configBad THEN
        _scaledWide := REAL_TO_LREAL(cfg.euMin)
            + (REAL_TO_LREAL(_clampedRaw) - REAL_TO_LREAL(cfg.rawMin))
            * (REAL_TO_LREAL(cfg.euMax) - REAL_TO_LREAL(cfg.euMin))
            / (REAL_TO_LREAL(cfg.rawMax) - REAL_TO_LREAL(cfg.rawMin));
        _scaledReal := LREAL_TO_REAL(LIMIT(LREAL#-3.402823E38, _scaledWide, LREAL#3.402823E38));
    ELSE
        _scaledReal := sts.value;
        sts.quality := E_IO_Quality.BAD;
    END_IF;
    sts.scaled := _scaledReal;

    // 4c. Optional first-order LPF. Pass-through when tau is 0.
    IF cfg.filterTau <> T#0MS THEN
        IF _reseedPending THEN
            _filter.Seed(value := REAL_TO_LREAL(_scaledReal));
        END_IF;
        _filter(
            fInput := _scaledReal,
            fDt    := _taskDtSec,
            fTau   := TIME_TO_REAL(cfg.filterTau) / 1000.0
        );
        _finalReal := LREAL_TO_REAL(_filter.fOutput);
    ELSE
        _finalReal := _scaledReal;
    END_IF;
END_IF;
_hasValidSample := TRUE;
_reseedPending := FALSE;
ELSE
    sts.clampedLow := FALSE;
    sts.clampedHigh := FALSE;
    sts.clampActive := FALSE;
END_IF;

sts.value := _finalReal;

// 5. Quality watchdog.
_tonBadQuality(
    IN := (_signalBad OR NOT (inpQuality = E_IO_Quality.GOOD OR inpQuality = E_IO_Quality.CLAMPED)) AND cfg.qualityFaultAfter > T#0MS,
    PT := cfg.qualityFaultAfter
);

// 6. Single-source-of-truth fault raise. See _RaiseActiveFault for priority.
_RaiseActiveFault();

// 7. Refresh shared header.
_UpdateHeader(header := sts.header, stateString := '', busy := FALSE);

// Pick the highest-severity active fault and raise it. Priority:
//   BadConfig (commissioning)
//   BadQuality (watchdog)
//   ClampHigh / ClampLow (if clampAsFault)
//
// If no rule applies the active fault (if any) is cleared so the device
// auto-recovers when the condition goes away.
METHOD PROTECTED _RaiseActiveFault
VAR
    code   : DINT;
    source : STRING(31);
    reason : STRING(79);
END_VAR
code := 0;

IF _configBad THEN
    code   := E_AnalogInput_Fault.BadConfig;
    source := 'CONFIG';
    reason := 'rawMin >= rawMax or euMin > euMax';
ELSIF _tonBadQuality.Q THEN
    code   := E_AnalogInput_Fault.BadQuality;
    source := 'QUALITY';
    reason := 'inpQuality stayed BAD past qualityFaultAfter';
ELSIF cfg.clampAsFault AND sts.clampedHigh THEN
    code   := E_AnalogInput_Fault.ClampHigh;
    source := 'CLAMP_H';
    reason := CONCAT('Raw reading above RawMax=', REAL_TO_STRING(cfg.rawMax));
ELSIF cfg.clampAsFault AND sts.clampedLow THEN
    code   := E_AnalogInput_Fault.ClampLow;
    source := 'CLAMP_L';
    reason := CONCAT('Raw reading below RawMin=', REAL_TO_STRING(cfg.rawMin));
END_IF;

IF code = 0 THEN
    IF IsFaulted() THEN
        _ClearFault();
    END_IF;
ELSE
    _Raise(
        code   := code,
        source := source,
        reason := reason
    );
END_IF;
END_METHOD

METHOD PROTECTED ResolveFaultString : STRING(79)
VAR_INPUT
    code : DINT;
END_VAR
CASE code OF
    0:
        ResolveFaultString := '';
    E_AnalogInput_Fault.BadQuality:
        ResolveFaultString := 'Signal quality BAD past configured timeout';
    E_AnalogInput_Fault.ClampLow:
        ResolveFaultString := 'Raw reading below RawMin';
    E_AnalogInput_Fault.ClampHigh:
        ResolveFaultString := 'Raw reading above RawMax';
    E_AnalogInput_Fault.BadConfig:
        ResolveFaultString := 'Invalid scaling range configured';
ELSE
    ResolveFaultString := CONCAT('AnalogInput fault ', DINT_TO_STRING(code));
END_CASE;
END_METHOD

// Owning-task application API: invalidate history when binding a different source.
// Call before supplying its first fresh sample; this is not a remote command.
METHOD PUBLIC ReassignInput
_hasValidSample := FALSE;
_reseedPending := TRUE;
sts.value := 0.0;
sts.scaled := 0.0;
sts.rawReal := 0.0;
sts.quality := E_IO_Quality.UNKNOWN;
sts.clampedLow := FALSE;
sts.clampedHigh := FALSE;
sts.clampActive := FALSE;
_tonBadQuality(IN := FALSE);
END_METHOD

END_FUNCTION_BLOCK

// ---- POUs/Utilities/FB_LPF_FirstOrder_IIR.TcPOU
// First-order IIR low-pass filter. Exponential smoothing of the form
//     y[n] = y[n-1] + alpha * (x[n] - y[n-1])
// with alpha = dt / (tau + dt). Tau is the 63.2 % rise-time constant.
//
// When dt or tau are effectively zero the filter passes the input through
// unchanged and raises bError. _prevOutput_sync persists across scans so the
// filter state carries between calls; it is ordinary non-retained state.
FUNCTION_BLOCK FB_LPF_FirstOrder_IIR
VAR_INPUT
    fInput  : LREAL;    // input sample
    fDt     : LREAL;    // time since previous call [s]
    fTau    : LREAL;    // time constant [s]
END_VAR
VAR_OUTPUT
    fOutput : LREAL;    // filtered output
    bError  : BOOL;     // TRUE when fDt or fTau were too small to filter
END_VAR
VAR
    _filtAlpha        : LREAL;
    _prevOutput_sync  : LREAL;
END_VAR

// Reject nonfinite values before they can poison retained recurrence history.
IF NOT F_IsFiniteLReal(value := _prevOutput_sync) THEN
    _prevOutput_sync := 0.0;
END_IF;
IF NOT F_IsFiniteLReal(value := fInput) OR NOT F_IsFiniteLReal(value := fDt) OR NOT F_IsFiniteLReal(value := fTau) THEN
    fOutput := _prevOutput_sync;
    bError := TRUE;
    RETURN;
END_IF;
// Preserve the documented finite zero/negative timing pass-through behavior.
IF fDt < 1E-38 OR fTau < 1E-38 THEN
    fOutput := fInput;
    bError  := TRUE;
    _prevOutput_sync := fOutput;
    RETURN;
END_IF;

bError := FALSE;

// Ratio form avoids overflow in tau + dt; weighted sum avoids x - previous.
IF fDt >= fTau THEN
    _filtAlpha := 1.0 / (1.0 + fTau / fDt);
ELSE
    _filtAlpha := fDt / fTau;
    _filtAlpha := _filtAlpha / (1.0 + _filtAlpha);
END_IF;
fOutput := (1.0 - _filtAlpha) * _prevOutput_sync + _filtAlpha * fInput;

_prevOutput_sync := fOutput;

// Explicit conditioning lifecycle reset, invoked only by the owning task.
// Invalid seeds leave existing history and output unchanged.
METHOD PUBLIC Seed : BOOL
VAR_INPUT value : LREAL; END_VAR
Seed := F_IsFiniteLReal(value := value);
IF NOT Seed THEN RETURN; END_IF;
_prevOutput_sync := value;
fOutput := value;
bError := FALSE;
END_METHOD

END_FUNCTION_BLOCK

// ---- POUs/IO/AnalogOutput/FB_AnalogOutput.TcPOU
// Generic analog output driver.
//
// Pipeline:
//   SetValue -> explicit command -> clamp to MinCv/MaxCv -> EU-to-raw
//   linear scaling -> UNION write (type chosen by cfg.outputType)
//
// Saved intent is restored only with cfg.restoreCommandOnRestart.
// Quality loss disarms output; recovery requires a fresh accepted command.
// ForceSafe and Reset inhibit output independent of the previous command.
//
{attribute 'OPC.UA.DA' := '1'}
FUNCTION_BLOCK FB_AnalogOutput EXTENDS FB_DeviceBase
VAR_INPUT
    {attribute 'OPC.UA.DA' := '1'}
    {attribute 'OPC.UA.DA.Access' := '1'}
    cfg        : ST_AnalogOutput_Cfg;
    {attribute 'OPC.UA.DA' := '0'}
    inpQuality : E_IO_Quality := E_IO_Quality.GOOD;
END_VAR

VAR_OUTPUT
    {attribute 'OPC.UA.DA' := '1'}
    {attribute 'OPC.UA.DA.Access' := '1'}
    outRaw : U_IoRaw_Out;
    {attribute 'OPC.UA.DA' := '1'}
    {attribute 'OPC.UA.DA.Access' := '1'}
    sts : ST_AnalogOutput_Sts;
END_VAR

VAR PERSISTENT
    // Saved intent (EU) and validity; durability depends on target persistent saving.
    {attribute 'OPC.UA.DA' := '0'}
    _savedCommand : REAL;
    {attribute 'OPC.UA.DA' := '0'}
    _savedCommandValid : BOOL;
END_VAR

VAR
    _configurationKnown : BOOL;
    _lastConfiguration : ST_AnalogOutput_Cfg;
    _requestSync : REAL; // Operating intent is never restored implicitly.
    _armed : BOOL;
    _commandReceived : BOOL;
    _startup : BOOL := TRUE;
    _forceSafe : BOOL;
    _safeRequested : BOOL;
    _qualityGood : BOOL;

    {attribute 'OPC.UA.DA' := '0'}
    _configBad     : BOOL;

    // Quality watchdog.
    {attribute 'OPC.UA.DA' := '0'}
    _tonBadQuality : TON;

    // Scratch values.
    {attribute 'OPC.UA.DA' := '0'}
    _clampedEu     : REAL;
    {attribute 'OPC.UA.DA' := '0'}
    _rawReal       : REAL;
    _rawWide       : LREAL;
END_VAR

_SyncConfiguration();
_ProcessOperatorCommands();
_qualityGood := inpQuality = E_IO_Quality.GOOD OR inpQuality = E_IO_Quality.CLAMPED;
IF _startup THEN
    _startup := FALSE;
    // A valid marker in a missing/backup image cannot authorize old operating intent.
    // A command accepted in this execution is fresh and does not depend on that image.
    IF NOT _commandReceived AND NOT THIS^._HasTrustedPersistentImage() THEN
        _savedCommandValid := FALSE;
    END_IF;
    IF NOT _commandReceived AND cfg.restoreCommandOnRestart AND _savedCommandValid THEN
        // Persistent data must be classified before it reaches floating operations.
        IF F_IsFiniteReal(_savedCommand) THEN
            _requestSync := _savedCommand;
            _armed := TRUE;
        ELSE
            _savedCommand := 0.0;
            _savedCommandValid := FALSE;
            _requestSync := 0.0;
            _armed := FALSE;
            _forceSafe := TRUE;
        END_IF;
    END_IF;
END_IF;
IF NOT _qualityGood THEN _armed := FALSE; END_IF;
// Validate every scan; live configuration changes cannot bypass validation.
// NaN/infinity classification uses bits; floating comparisons can trap on the PLC.
_configBad := NOT (F_IsFiniteReal(cfg.safeRaw) AND F_IsFiniteReal(cfg.euMin) AND F_IsFiniteReal(cfg.euMax) AND F_IsFiniteReal(cfg.rawMin) AND F_IsFiniteReal(cfg.rawMax) AND F_IsFiniteReal(cfg.minCv) AND F_IsFiniteReal(cfg.maxCv));
IF NOT _configBad THEN
    _configBad := (NOT cfg.useRawValue AND (cfg.euMin >= cfg.euMax OR cfg.rawMin >= cfg.rawMax OR cfg.minCv > cfg.maxCv))
                  OR NOT ((cfg.euMin >= -1.0E30 AND cfg.euMin <= 1.0E30) AND (cfg.euMax >= -1.0E30 AND cfg.euMax <= 1.0E30) AND (cfg.rawMin >= -1.0E30 AND cfg.rawMin <= 1.0E30) AND (cfg.rawMax >= -1.0E30 AND cfg.rawMax <= 1.0E30) AND (cfg.minCv >= -1.0E30 AND cfg.minCv <= 1.0E30) AND (cfg.maxCv >= -1.0E30 AND cfg.maxCv <= 1.0E30));
END_IF;
_configBad := _configBad OR NOT (cfg.outputType = __SYSTEM.TYPE_CLASS.TYPE_INT OR cfg.outputType = __SYSTEM.TYPE_CLASS.TYPE_UINT OR cfg.outputType = __SYSTEM.TYPE_CLASS.TYPE_WORD OR cfg.outputType = __SYSTEM.TYPE_CLASS.TYPE_DINT OR cfg.outputType = __SYSTEM.TYPE_CLASS.TYPE_UDINT OR cfg.outputType = __SYSTEM.TYPE_CLASS.TYPE_DWORD OR cfg.outputType = __SYSTEM.TYPE_CLASS.TYPE_REAL);

sts.unit       := cfg.unit;
sts.quality    := inpQuality;
sts.commanded  := _requestSync;

// 2. Clamp the command in EU space.
sts.clampedLow  := FALSE;
sts.clampedHigh := FALSE;
_clampedEu         := _requestSync;

IF NOT _configBad AND NOT cfg.useRawValue THEN
    IF _clampedEu < cfg.minCv THEN
        _clampedEu        := cfg.minCv;
        sts.clampedLow := TRUE;
    ELSIF _clampedEu > cfg.maxCv THEN
        _clampedEu         := cfg.maxCv;
        sts.clampedHigh := TRUE;
    END_IF;
END_IF;
sts.clampActive := sts.clampedLow OR sts.clampedHigh;
// sts.value is updated only when the command is actually applied.

// Scale with wide intermediates, then bound before narrowing to REAL.
IF _configBad THEN
    _rawWide := 0.0;
ELSIF cfg.useRawValue THEN
    _rawWide := REAL_TO_LREAL(_clampedEu);
ELSE
    _rawWide := REAL_TO_LREAL(cfg.rawMin)
              + (REAL_TO_LREAL(cfg.rawMax) - REAL_TO_LREAL(cfg.rawMin))
                * ((REAL_TO_LREAL(_clampedEu) - REAL_TO_LREAL(cfg.euMin))
                / (REAL_TO_LREAL(cfg.euMax) - REAL_TO_LREAL(cfg.euMin)));
END_IF;
_rawReal := LREAL_TO_REAL(LIMIT(LREAL#-3.402823E38, _rawWide, LREAL#3.402823E38));
// Raw status is published after output policy.

// Fault decisions precede output application.
_tonBadQuality(IN := NOT _qualityGood AND cfg.qualityFaultAfter > T#0MS, PT := cfg.qualityFaultAfter);
_RaiseActiveFault();
IF IsFaulted() THEN _armed := FALSE; END_IF;
IF _forceSafe OR IsFaulted() OR (_qualityGood AND NOT _armed) OR (NOT _qualityGood AND NOT cfg.holdOnBadQuality) THEN
    IF F_IsFiniteReal(cfg.safeRaw) THEN _rawReal := cfg.safeRaw;
    ELSE _rawReal := 0.0; END_IF;
    sts.value := 0.0; // EU value is unavailable when applying a raw fallback; see outputInhibited.
ELSIF NOT _qualityGood THEN
    _rawReal := sts.rawReal;
ELSE
    sts.value := _clampedEu;
END_IF;
sts.outputInhibited := NOT _armed OR _forceSafe OR IsFaulted();
// Classify before any LIMIT comparison or conversion, including held terminal state.
IF NOT F_IsFiniteReal(_rawReal) THEN _rawReal := 0.0; END_IF;
// Conversion is bounded to the representable terminal range before any cast.
CASE cfg.outputType OF
    __SYSTEM.TYPE_CLASS.TYPE_INT:   _rawReal := LIMIT(-32768.0, _rawReal, 32767.0);
    __SYSTEM.TYPE_CLASS.TYPE_UINT, __SYSTEM.TYPE_CLASS.TYPE_WORD: _rawReal := LIMIT(0.0, _rawReal, 65535.0);
    __SYSTEM.TYPE_CLASS.TYPE_DINT: _rawReal := LIMIT(-2147483648.0, _rawReal, 2147483520.0);
    __SYSTEM.TYPE_CLASS.TYPE_UDINT, __SYSTEM.TYPE_CLASS.TYPE_DWORD: _rawReal := LIMIT(0.0, _rawReal, 4294967040.0);
END_CASE;
outRaw.dw := 0; // Clear upper bytes when writing a 16-bit member.
CASE cfg.outputType OF
    __SYSTEM.TYPE_CLASS.TYPE_INT: outRaw.nInt := REAL_TO_INT(_rawReal);
    __SYSTEM.TYPE_CLASS.TYPE_UINT: outRaw.ui := REAL_TO_UINT(_rawReal);
    __SYSTEM.TYPE_CLASS.TYPE_WORD: outRaw.w := REAL_TO_WORD(_rawReal);
    __SYSTEM.TYPE_CLASS.TYPE_DINT: outRaw.di := REAL_TO_DINT(_rawReal);
    __SYSTEM.TYPE_CLASS.TYPE_UDINT: outRaw.udi := REAL_TO_UDINT(_rawReal);
    __SYSTEM.TYPE_CLASS.TYPE_DWORD: outRaw.dw := REAL_TO_DWORD(_rawReal);
    __SYSTEM.TYPE_CLASS.TYPE_REAL: outRaw.fReal := _rawReal;
ELSE
    outRaw.dw := 0;
END_CASE;
sts.rawReal := _rawReal;

_safeRequested := FALSE; // consumed after applying outputs

// 7. Refresh shared header.
_UpdateHeader(header := sts.header, stateString := '', busy := FALSE);

METHOD PUBLIC SetValue : E_RpcMethodResponse
VAR_INPUT
    rValue     : REAL;
    eRequester : E_Requester := E_Requester.PROG;
END_VAR
// Reject invalid identity before any command-specific mutation.
SetValue := F_ValidateRequester(eRequester := eRequester, bSourceLocked := FALSE, bFaulted := FALSE);
IF SetValue <> E_RpcMethodResponse.ACCEPTED THEN RETURN; END_IF;
_SyncConfiguration();
IF _safeRequested THEN
    SetValue := E_RpcMethodResponse.REJECTED_INTERLOCKED;
    RETURN;
END_IF;
IF NOT F_IsFiniteReal(rValue) THEN
    SetValue := E_RpcMethodResponse.REJECTED_INVALID_PARAMETER;
    RETURN;
END_IF;
SetValue := F_ValidateRequester(
    eRequester    := eRequester,
    bSourceLocked := bSourceLockedToProg,
    bFaulted      := IsFaulted()
);

IF SetValue <> E_RpcMethodResponse.ACCEPTED THEN
    RETURN;
END_IF;

_requestSync := rValue;
_savedCommand := _requestSync;
_savedCommandValid := TRUE;
_armed := TRUE;
_commandReceived := TRUE;
_forceSafe := FALSE;
_AcceptCommand(eRequester := eRequester);
END_METHOD

// Priority chain for AnalogOutput faults:
//   BadConfig > BadQuality > ClampHigh > ClampLow
METHOD PROTECTED _RaiseActiveFault
VAR
    code   : DINT;
    source : STRING(31);
    reason : STRING(79);
END_VAR
code := 0;

IF _configBad THEN
    code   := E_AnalogOutput_Fault.BadConfig;
    source := 'CONFIG';
    reason := 'euMin >= euMax or rawMin > rawMax';
ELSIF _tonBadQuality.Q THEN
    code   := E_AnalogOutput_Fault.BadQuality;
    source := 'QUALITY';
    reason := 'inpQuality stayed BAD past qualityFaultAfter';
ELSIF _armed AND cfg.clampAsFault AND sts.clampedHigh THEN
    code   := E_AnalogOutput_Fault.ClampHigh;
    source := 'CLAMP_H';
    reason := CONCAT('Command clamped at MaxCv=', REAL_TO_STRING(cfg.maxCv));
ELSIF _armed AND cfg.clampAsFault AND sts.clampedLow THEN
    code   := E_AnalogOutput_Fault.ClampLow;
    source := 'CLAMP_L';
    reason := CONCAT('Command clamped at MinCv=', REAL_TO_STRING(cfg.minCv));
END_IF;

IF code = 0 THEN
    // Output faults latch until Reset; configuration/quality recovery cannot restart them.
ELSE
    _Raise(
        code   := code,
        source := source,
        reason := reason
    );
END_IF;
END_METHOD

METHOD PROTECTED ResolveFaultString : STRING(79)
VAR_INPUT
    code : DINT;
END_VAR
CASE code OF
    0:
        ResolveFaultString := '';
    E_AnalogOutput_Fault.BadQuality:
        ResolveFaultString := 'Output quality BAD past configured timeout';
    E_AnalogOutput_Fault.ClampLow:
        ResolveFaultString := 'Command clamped at MinCv';
    E_AnalogOutput_Fault.ClampHigh:
        ResolveFaultString := 'Command clamped at MaxCv';
    E_AnalogOutput_Fault.BadConfig:
        ResolveFaultString := 'Invalid scaling range configured';
ELSE
    ResolveFaultString := CONCAT('AnalogOutput fault ', DINT_TO_STRING(code));
END_CASE;
END_METHOD

{attribute 'TcRpcEnable' := '1'}
METHOD PUBLIC OperatorSetValue : E_RpcMethodResponse
VAR_INPUT
    requestId : ULINT;
    rValue : REAL;
END_VAR
OperatorSetValue := _operatorMailbox.Submit(requestId := requestId, command := E_OperatorCommand.SetValue, value := rValue);
END_METHOD

